// SIMATIC STEP 7 (V5.x) project jiayao
// CPU: CPU 315-2 DP
// station: P_ADR_BUS
// station: 硬件
// station: SIMATIC 300(1)(1)
// program: S7 程序(1)

SYMBOL_TABLE
"DB1"	DB 1	DB 1
"DB2"	DB 2	DB 2
"配药"	FC 1	FC 1
"计量泵程序"	FC 2	FC 2
"自动曝气"	FC 3	FC 3
"自动出药"	FC 4	FC 4
"时间转换程序"	FC 6	FC 6
"模拟液位"	FC 7	FC 7
"报警"	FC 8	FC 8
"TIM_S5TI"	FC 40	FC 40	// IEC Time to S5 Time
"SCALE"	FC 105	FC 105	// Scaling Values
"1池远程本地"	I 0.0	BOOL
"1池进药阀开到位"	I 0.1	BOOL
"1池进药阀关到位"	I 0.2	BOOL
"1池进水阀开到位"	I 0.3	BOOL
"1池进水阀关到位"	I 0.4	BOOL
"1池气阀开到位"	I 0.5	BOOL
"1池气阀关到位"	I 0.6	BOOL
"1池出药阀开到位"	I 0.7	BOOL
"1池出药阀关到位"	I 1.0	BOOL
"2池远程本地"	I 1.1	BOOL
"2池进药阀开到位"	I 1.2	BOOL
"2池进药阀关到位"	I 1.3	BOOL
"2池进水阀开到位"	I 1.4	BOOL
"2池进水阀关到位"	I 1.5	BOOL
"2池气阀开到位"	I 1.6	BOOL
"2池气阀关到位"	I 1.7	BOOL
"2池出药阀开到位"	I 2.0	BOOL
"2池出药阀关到位"	I 2.1	BOOL
"1号曝气泵远程本地"	I 2.2	BOOL
"1号曝气泵运行状态"	I 2.3	BOOL
"1号曝气泵热继故障"	I 2.4	BOOL
"2号曝气泵远程本地"	I 2.5	BOOL
"2号曝气泵运行状态"	I 2.6	BOOL
"2号曝气泵热继故障"	I 2.7	BOOL
"补水阀开到位"	I 3.0	BOOL
"新系统变频远程"	I 3.2	BOOL
"老系统变频远程"	I 3.3	BOOL
"1池自动遥控"	M 0.0	BOOL
"1池进药阀遥控开阀"	M 0.1	BOOL
"1池进药阀遥控关阀"	M 0.2	BOOL
"1池进水阀遥控开阀"	M 0.3	BOOL
"1池进水阀遥控关阀"	M 0.4	BOOL
"1池曝气阀遥控开阀"	M 0.5	BOOL
"1池曝气阀遥控关阀"	M 0.6	BOOL
"1池出药阀遥控开阀"	M 0.7	BOOL
"1池出药阀遥控关阀"	M 1.0	BOOL
"2池自动遥控"	M 1.1	BOOL
"2池进药阀遥控开阀"	M 1.2	BOOL
"2池进药阀遥控关阀"	M 1.3	BOOL
"2池进水阀遥控开阀"	M 1.4	BOOL
"2池进水阀遥控关阀"	M 1.5	BOOL
"2池进气阀遥控开阀"	M 1.6	BOOL
"2池进气阀遥控关阀"	M 1.7	BOOL
"2池出药阀遥控开阀"	M 2.0	BOOL
"2池出药阀遥控关阀"	M 2.1	BOOL
"1号曝气泵自动遥控"	M 2.2	BOOL
"1号曝气泵遥控启动"	M 2.3	BOOL
"1号曝气泵遥控停止"	M 2.4	BOOL
"2号曝气泵自动遥控"	M 2.5	BOOL
"2号曝气泵遥控启动"	M 2.6	BOOL
"2号曝气泵遥控停止"	M 2.7	BOOL
"新系统变频遥控自动"	M 3.0	BOOL
"新系统变频遥控启动"	M 3.1	BOOL
"新系统变频遥控停止"	M 3.2	BOOL
"老系统变频遥控自动"	M 3.3	BOOL
"老系统变频遥控启动"	M 3.4	BOOL
"老系统变频遥控停止"	M 3.5	BOOL
"1池空池"	M 3.6	BOOL
"2池空池"	M 3.7	BOOL
"1池确认配药"	M 4.0	BOOL
"2池确认配药"	M 4.1	BOOL
"1池取消配药"	M 4.2	BOOL
"2池取消配药"	M 4.3	BOOL
"1池开始配药"	M 4.4	BOOL
"2池开始配药"	M 4.5	BOOL
"补水阀自动遥控"	M 4.6	BOOL
"1池自动曝气系统故障"	M 4.7	BOOL
"1池气阀自动开关"	M 6.2	BOOL
"2池气阀自动开关"	M 6.3	BOOL
"配药池1号出药阀自动运行"	M 6.4	BOOL
"配药池2号出药阀自动运行"	M 6.5	BOOL
"补水阀遥控开"	M 6.6	BOOL
"补水阀遥控关"	M 6.7	BOOL
"1池气阀自动开关(延时关)"	M 7.2	BOOL
"2池气阀自动开关(延时关)"	M 7.3	BOOL
"补水阀自动开关"	M 8.6	BOOL
"1号曝气泵自动运行"	M 8.7	BOOL
"2号曝气泵自动运行"	M 9.0	BOOL
"曝气泵切换"	M 11.2	BOOL
"2.3I下降沿"	M 13.0	BOOL
"2.6I下降沿"	M 13.3	BOOL
"FC105块极性选择0为单极性"	M 15.0	BOOL
"4.4m上升沿"	M 17.1	BOOL
"1池有药"	M 17.2	BOOL
"4.5m上升沿"	M 17.3	BOOL
"2池有药"	M 17.4	BOOL
"46.6M上升沿"	M 17.5	BOOL
"47.1M上升沿"	M 17.6	BOOL
"45.0M上升沿"	M 17.7	BOOL
"1号气泵就绪"	M 18.0	BOOL
"45.1m上升沿"	M 18.1	BOOL
"2号气泵就绪"	M 18.2	BOOL
"1池计时器:运行时间上升沿"	M 18.5	BOOL
"2池计时器:运行时间上升沿"	M 18.7	BOOL
"T1计时器"	M 19.0	BOOL
"T6计时器"	M 19.1	BOOL
"1池加药阀自动运行"	M 19.2	BOOL
"1池加水阀自动运行"	M 19.3	BOOL
"2池加药阀自动运行"	M 19.4	BOOL
"2池加水阀自动运行"	M 19.5	BOOL
"1池自动曝气就绪"	M 45.0	BOOL
"2池自动曝气就绪"	M 45.1	BOOL
"2池自动曝气系统故障"	M 45.2	BOOL
"1池进药阀开故障"	M 45.3	BOOL
"1池进药阀关故障"	M 45.4	BOOL
"补水阀故障"	M 45.5	BOOL
"1池曝气请求"	M 45.6	BOOL
"2池曝气请求"	M 45.7	BOOL
"1池自动出药就绪"	M 46.0	BOOL
"1池自动出药系统故障"	M 46.1	BOOL
"1池出药阀故障"	M 46.2	BOOL
"2池自动出药系统故障"	M 46.3	BOOL
"2池自动出药就绪"	M 46.4	BOOL
"2池出药阀故障"	M 46.5	BOOL
"1池配药系统就绪"	M 46.6	BOOL
"1池配药系统故障"	M 46.7	BOOL
"2池配药系统故障"	M 47.0	BOOL
"2池配药系统就绪"	M 47.1	BOOL
"1池曝气阀故障"	M 47.2	BOOL
"2池曝气阀故障"	M 47.3	BOOL
"新系统自动运行"	M 47.4	BOOL
"1池配药"	M 47.5	BOOL
"2池配药"	M 47.6	BOOL
"老系统自动运行"	M 47.7	BOOL
"新系统变频器故障"	M 48.0	BOOL
"老系统变频器故障"	M 48.1	BOOL
"1池进药阀故障"	M 48.2	BOOL
"1池进水阀故障"	M 48.3	BOOL
"2池进药阀故障"	M 48.4	BOOL
"2池进水阀故障"	M 48.5	BOOL
"1池进水阀开故障"	M 48.6	BOOL
"1池进水阀关故障"	M 48.7	BOOL
"1池气阀开故障"	M 49.0	BOOL
"1池气阀关故障"	M 49.1	BOOL
"1池出药阀开故障"	M 49.2	BOOL
"1池出药阀关故障"	M 49.3	BOOL
"2池进药阀开故障"	M 49.4	BOOL
"2池进药阀关故障"	M 49.5	BOOL
"2池进水阀开故障"	M 49.6	BOOL
"2池进水阀关故障"	M 49.7	BOOL
"2池气阀开故障"	M 50.0	BOOL
"2池气阀关故障"	M 50.1	BOOL
"2池出药阀开故障"	M 50.2	BOOL
"2池出药阀关故障"	M 50.3	BOOL
"1号曝气泵运行故障"	M 50.4	BOOL
"2号曝气泵运行故障"	M 50.5	BOOL
"1池液位故障"	M 50.6	BOOL
"1池液位断线"	M 50.7	BOOL
"2池液位故障"	M 51.0	BOOL
"2池液位断线"	M 51.1	BOOL
"原液池液位故障"	M 51.2	BOOL
"原液池液位断线"	M 51.3	BOOL
"新系统瞬时流量下限报警"	M 51.4	BOOL	// 没用，组态已取暂留
"老系统瞬时流量下限报警"	M 51.5	BOOL	// 没用，组态已取暂留
"触摸屏消音"	M 51.6	BOOL
"COMPLETE RESTART"	OB 100	OB 100	// Complete Restart
"PROG_ERR"	OB 121	OB 121	// Programming Error
"1池进药阀开关"	Q 0.0	BOOL
"1池进水阀开关"	Q 0.1	BOOL
"1池气阀开关"	Q 0.2	BOOL
"配药池1号出药阀开关"	Q 0.3	BOOL
"2池进药阀开关"	Q 0.4	BOOL
"2池进水阀开关"	Q 0.5	BOOL
"2池气阀开关"	Q 0.6	BOOL
"配药池2号出药阀开关"	Q 0.7	BOOL
"曝气泵1号启停"	Q 1.0	BOOL
"曝气泵2号启停"	Q 1.1	BOOL
"补水阀开关"	Q 1.2	BOOL
"新系统变频启停"	Q 1.3	BOOL
"老系统变频启停"	Q 1.4	BOOL
"嗡鸣器"	Q 1.5	BOOL
"1池计时器"	T 1	TIMER
"2池计时器"	T 6	TIMER
"2池达到加药后液位"	T 7	TIMER
"2池达到加水后液位"	T 8	TIMER
"1池进药阀开故障延时"	T 9	TIMER
"1池进药阀关故障延时"	T 10	TIMER
"1池进水阀开故障延时"	T 11	TIMER
"1池进水阀关故障延时"	T 12	TIMER
"1池气阀开故障延时"	T 13	TIMER
"1池气阀关故障延时"	T 14	TIMER
"1池出药阀开故障延时"	T 15	TIMER
"1池出药阀关故障延时"	T 16	TIMER
"2池进药阀开故障延时"	T 17	TIMER
"2池进药阀关故障延时"	T 18	TIMER
"2池进水阀开故障延时"	T 19	TIMER
"2池进水阀关故障延时"	T 20	TIMER
"2池气阀开故障延时"	T 21	TIMER
"2池气阀关故障延时"	T 22	TIMER
"2池出药阀开故障延时"	T 23	TIMER
"2池出药阀关故障延时"	T 24	TIMER
"补水阀开故障延时"	T 25	TIMER
"1号曝气泵运行故障延时"	T 26	TIMER
"2号曝气泵运行故障延时"	T 27	TIMER
"1池达到加药后液位"	T 37	TIMER
"1池达到加水后液位"	T 38	TIMER
"1池曝气运行时间"	T 41	TIMER
"2池曝气运行时间"	T 42	TIMER
"新系统出药流量低延时"	T 44	TIMER
"老系统出药流量低延时"	T 45	TIMER
"1池延时断开"	T 46	TIMER
"2池延时断开"	T 47	TIMER
"1池空池延时"	T 48	TIMER
"2池空池延时"	T 49	TIMER
END_SYMBOL_TABLE

FUNCTION "配药" : VOID	// FC 1
//配药
VERSION : 0.1
BEGIN
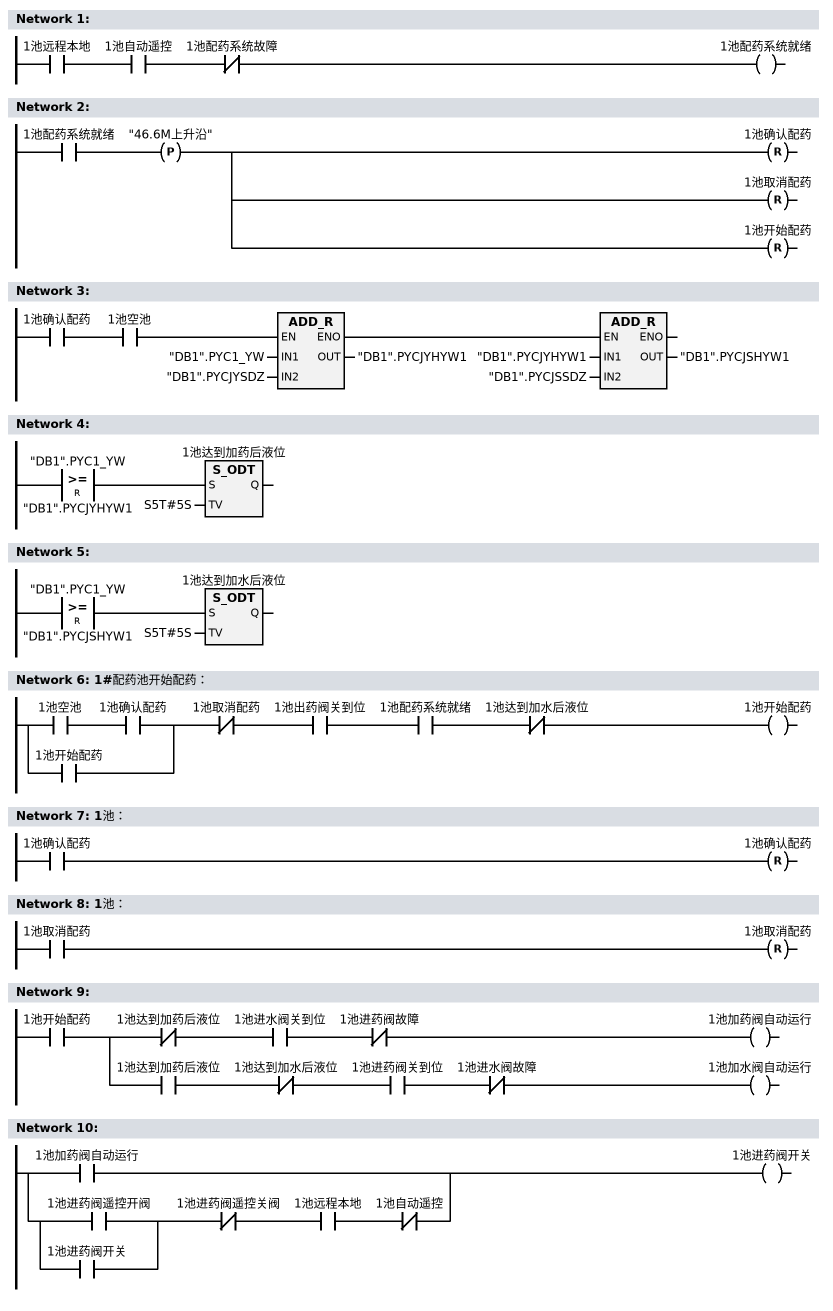
NETWORK
TITLE =
//1#配药池：配药就绪检测
      A     "1池远程本地";
      A     "1池自动遥控";
      AN    "1池配药系统故障";
      =     "1池配药系统就绪";
NETWORK
TITLE =
//1#配药池配药就绪后复位1#配药池确认、1#配药池取消配药和1#配药池开始配药
      A     "1池配药系统就绪";
      FP    "46.6M上升沿";
      R     "1池确认配药";
      R     "1池取消配药";
      R     "1池开始配药";
NETWORK
TITLE =
//1#配药池确认配药和1#配药池空池时，用1#配药池液位加上加药量设定得到1#配药池加药
//
//后的液位，用1#配药池加药后的液位加上加水量设定得到1#配药池加水后液位
      A(;
      A     "1池确认配药";
      A     "1池空池";
      JNB   _001;
      L     "DB1".PYC1_YW;
      L     "DB1".PYCJYSDZ;
      +R;
      T     "DB1".PYCJYHYW1;
      AN    OV;
      SAVE;
      CLR;
_001: A     BR;
      );
      JNB   _002;
      L     "DB1".PYCJYHYW1;
      L     "DB1".PYCJSSDZ;
      +R;
      T     "DB1".PYCJSHYW1;
_002: NOP   0;
NETWORK
TITLE =
//1#配药池液位大于等于1#加药后液位设定，延时5秒
      A(;
      L     "DB1".PYC1_YW;
      L     "DB1".PYCJYHYW1;
      >=R;
      );
      L     S5T#5S;
      SD    "1池达到加药后液位";
      NOP   0;
      NOP   0;
      NOP   0;
      NOP   0;
NETWORK
TITLE =
//1#配药池液位大于等于1#加水后液位设定，延时5秒
      A(;
      L     "DB1".PYC1_YW;
      L     "DB1".PYCJSHYW1;
      >=R;
      );
      L     S5T#5S;
      SD    "1池达到加水后液位";
      NOP   0;
      NOP   0;
      NOP   0;
      NOP   0;
NETWORK
TITLE = 1#配药池开始配药：
//
//1#配药池空池、1#配药池确认配药、1#配药池没有取消配药、1#配药池出药阀关到位、1#配
//
//药池系统就绪、1#配药池没到加水后液位，1#配药池开始配药
      A(;
      A     "1池空池";
      A     "1池确认配药";
      O     "1池开始配药";
      );
      AN    "1池取消配药";
      A     "1池出药阀关到位";
      A     "1池配药系统就绪";
      AN    "1池达到加水后液位";
      =     "1池开始配药";
NETWORK
TITLE = 1池：
//1#配药池确认配药复位
      A     "1池确认配药";
      R     "1池确认配药";
NETWORK
TITLE = 1池：
//1#配药池取消配药复位
      A     "1池取消配药";
      R     "1池取消配药";
NETWORK
TITLE =
//1#配药池开始配药，1#配药池没有达到加药后液位、1#配药池进水阀门关到位和1#配药池进
//
//药阀门无故障，1#配药池加药阀门自动运行。
//
//1#配药池开始配药，1#配药池达到加药后液位、1#配药池没有达到加水后液位、1#配药池进
//
//药阀门关到位和1#配药池进水阀门无故障，1#配药池加水阀门自动运行。
      A     "1池开始配药";
      =     L 0.0;
      A     L 0.0;
      AN    "1池达到加药后液位";
      A     "1池进水阀关到位";
      AN    "1池进药阀故障";
      =     "1池加药阀自动运行";
      A     L 0.0;
      A     "1池达到加药后液位";
      AN    "1池达到加水后液位";
      A     "1池进药阀关到位";
      AN    "1池进水阀故障";
      =     "1池加水阀自动运行";
NETWORK
TITLE =
//1#配药池进药阀自动控制和遥控控制
      O     "1池加药阀自动运行";
      O;
      A(;
      O     "1池进药阀遥控开阀";
      O     "1池进药阀开关";
      );
      AN    "1池进药阀遥控关阀";
      A     "1池远程本地";
      AN    "1池自动遥控";
      =     "1池进药阀开关";
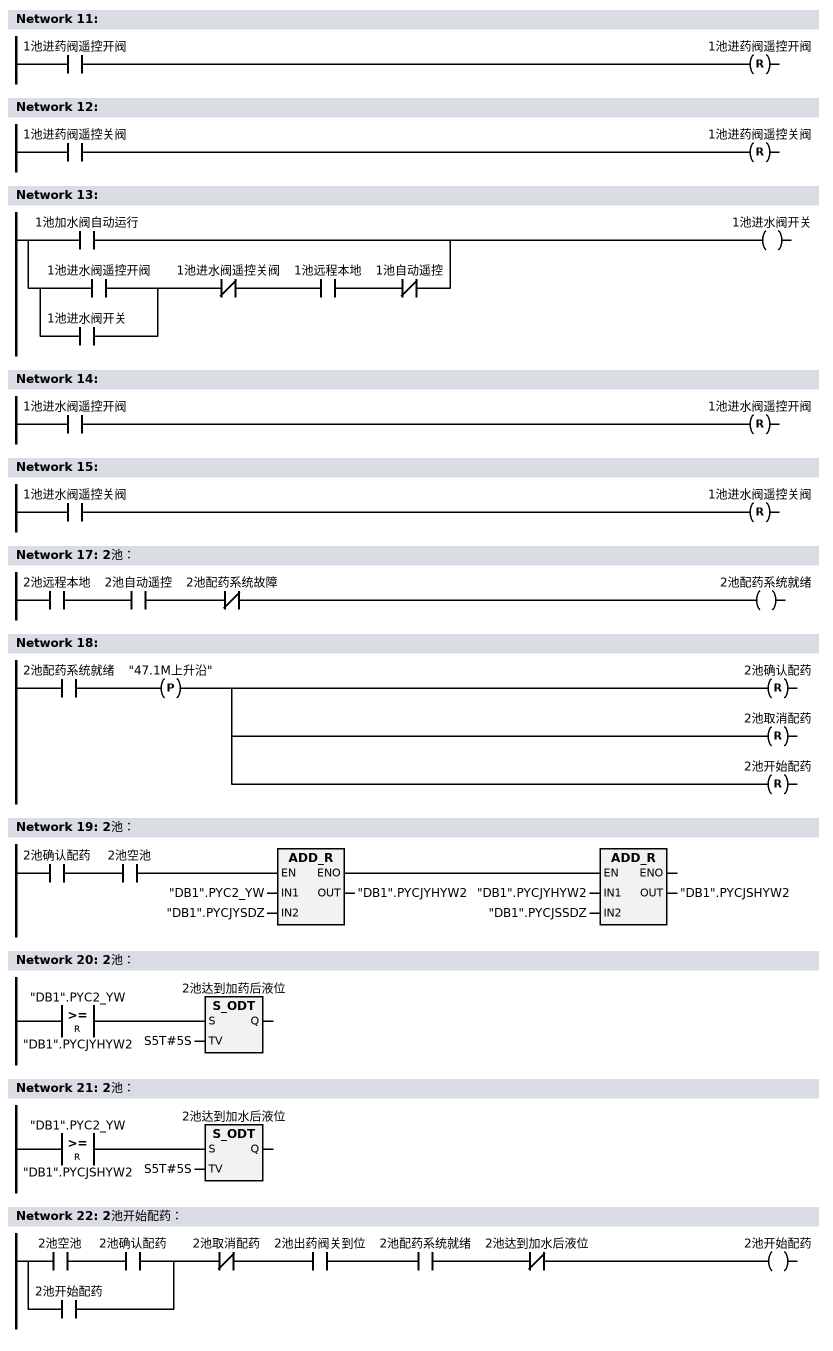
NETWORK
TITLE =
//1#配药池进药阀遥控开复位
      A     "1池进药阀遥控开阀";
      R     "1池进药阀遥控开阀";
NETWORK
TITLE =
//1#配药池进药阀遥控关复位
      A     "1池进药阀遥控关阀";
      R     "1池进药阀遥控关阀";
NETWORK
TITLE =
//1#配药池进水阀自动控制和遥控控制
      O     "1池加水阀自动运行";
      O;
      A(;
      O     "1池进水阀遥控开阀";
      O     "1池进水阀开关";
      );
      AN    "1池进水阀遥控关阀";
      A     "1池远程本地";
      AN    "1池自动遥控";
      =     "1池进水阀开关";
NETWORK
TITLE =
//1#配药池进水阀遥控开复位
      A     "1池进水阀遥控开阀";
      R     "1池进水阀遥控开阀";
NETWORK
TITLE =
//1#配药池进水阀遥控关复位
      A     "1池进水阀遥控关阀";
      R     "1池进水阀遥控关阀";
NETWORK
TITLE =
NETWORK
TITLE = 2池：
//2#配药池：配药就绪检测
      A     "2池远程本地";
      A     "2池自动遥控";
      AN    "2池配药系统故障";
      =     "2池配药系统就绪";
NETWORK
TITLE =
//2#配药池配药就绪后复位2#配药池确认、2#配药池取消配药和2#配药池开始配药
      A     "2池配药系统就绪";
      FP    "47.1M上升沿";
      R     "2池确认配药";
      R     "2池取消配药";
      R     "2池开始配药";
NETWORK
TITLE = 2池：
//2#配药池确认配药和2#配药池空池时，用2#配药池液位加上加药量设定得到2#配药池加药
//
//后的液位，用2#配药池加药后的液位加上加水量设定得到2#配药池加水后液位
      A(;
      A     "2池确认配药";
      A     "2池空池";
      JNB   _003;
      L     "DB1".PYC2_YW;
      L     "DB1".PYCJYSDZ;
      +R;
      T     "DB1".PYCJYHYW2;
      AN    OV;
      SAVE;
      CLR;
_003: A     BR;
      );
      JNB   _004;
      L     "DB1".PYCJYHYW2;
      L     "DB1".PYCJSSDZ;
      +R;
      T     "DB1".PYCJSHYW2;
_004: NOP   0;
NETWORK
TITLE = 2池：
//2#配药池液位大于等于2#加药后液位设定，延时5秒
      A(;
      L     "DB1".PYC2_YW;
      L     "DB1".PYCJYHYW2;
      >=R;
      );
      L     S5T#5S;
      SD    "2池达到加药后液位";
      NOP   0;
      NOP   0;
      NOP   0;
      NOP   0;
NETWORK
TITLE = 2池：
//2#配药池液位大于等于2#加水后液位设定，延时5秒
      A(;
      L     "DB1".PYC2_YW;
      L     "DB1".PYCJSHYW2;
      >=R;
      );
      L     S5T#5S;
      SD    "2池达到加水后液位";
      NOP   0;
      NOP   0;
      NOP   0;
      NOP   0;
NETWORK
TITLE = 2池开始配药：
//2#配药池空池、2#配药池确认配药、2#配药池没有取消配药、2#配药池出药阀关到位、2#配
//
//药池系统就绪、2#配药池没到加水后液位，2#配药池开始配药
      A(;
      A     "2池空池";
      A     "2池确认配药";
      O     "2池开始配药";
      );
      AN    "2池取消配药";
      A     "2池出药阀关到位";
      A     "2池配药系统就绪";
      AN    "2池达到加水后液位";
      =     "2池开始配药";
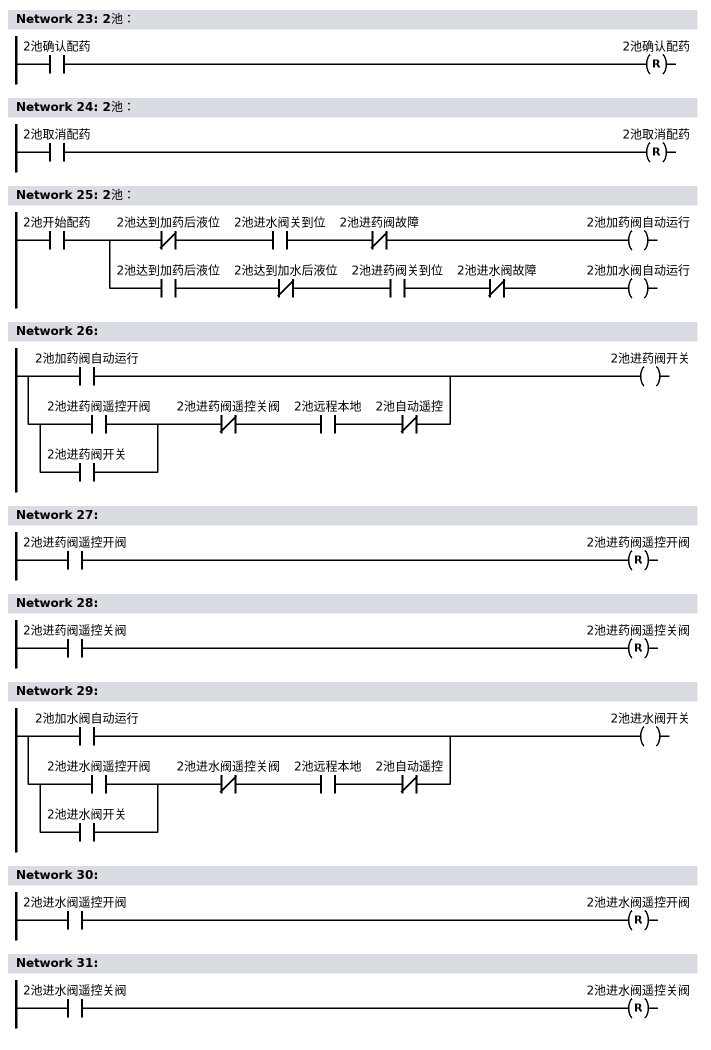
NETWORK
TITLE = 2池：
//2#配药池确认配药复位
      A     "2池确认配药";
      R     "2池确认配药";
NETWORK
TITLE = 2池：
//2#配药池取消配药复位
      A     "2池取消配药";
      R     "2池取消配药";
NETWORK
TITLE = 2池：
//2#配药池开始配药，2#配药池没有达到加药后液位、2#配药池进水阀门关到位和2#配药池进
//
//药阀门无故障，2#配药池加药阀门自动运行。
//
//2#配药池开始配药，2#配药池达到加药后液位、2#配药池没有达到加水后液位、2#配药池进
//
//药阀门关到位和2#配药池进水阀门无故障，2#配药池加水阀门自动运行
      A     "2池开始配药";
      =     L 0.0;
      A     L 0.0;
      AN    "2池达到加药后液位";
      A     "2池进水阀关到位";
      AN    "2池进药阀故障";
      =     "2池加药阀自动运行";
      A     L 0.0;
      A     "2池达到加药后液位";
      AN    "2池达到加水后液位";
      A     "2池进药阀关到位";
      AN    "2池进水阀故障";
      =     "2池加水阀自动运行";
NETWORK
TITLE =
//2#配药池进药阀自动控制和遥控控制
      O     "2池加药阀自动运行";
      O;
      A(;
      O     "2池进药阀遥控开阀";
      O     "2池进药阀开关";
      );
      AN    "2池进药阀遥控关阀";
      A     "2池远程本地";
      AN    "2池自动遥控";
      =     "2池进药阀开关";
NETWORK
TITLE =
//2#配药池进药阀遥控开复位
      A     "2池进药阀遥控开阀";
      R     "2池进药阀遥控开阀";
NETWORK
TITLE =
//2#配药池进药阀遥控关复位
      A     "2池进药阀遥控关阀";
      R     "2池进药阀遥控关阀";
NETWORK
TITLE =
//2#配药池进水阀自动控制和遥控控制
      O     "2池加水阀自动运行";
      O;
      A(;
      O     "2池进水阀遥控开阀";
      O     "2池进水阀开关";
      );
      AN    "2池进水阀遥控关阀";
      A     "2池远程本地";
      AN    "2池自动遥控";
      =     "2池进水阀开关";
NETWORK
TITLE =
//2#配药池进水阀遥控开复位
      A     "2池进水阀遥控开阀";
      R     "2池进水阀遥控开阀";
NETWORK
TITLE =
//2#配药池进水阀遥控关复位
      A     "2池进水阀遥控关阀";
      R     "2池进水阀遥控关阀";
END_FUNCTION

FUNCTION "计量泵程序" : VOID	// FC 2
//计量泵程序
VERSION : 0.1
BEGIN
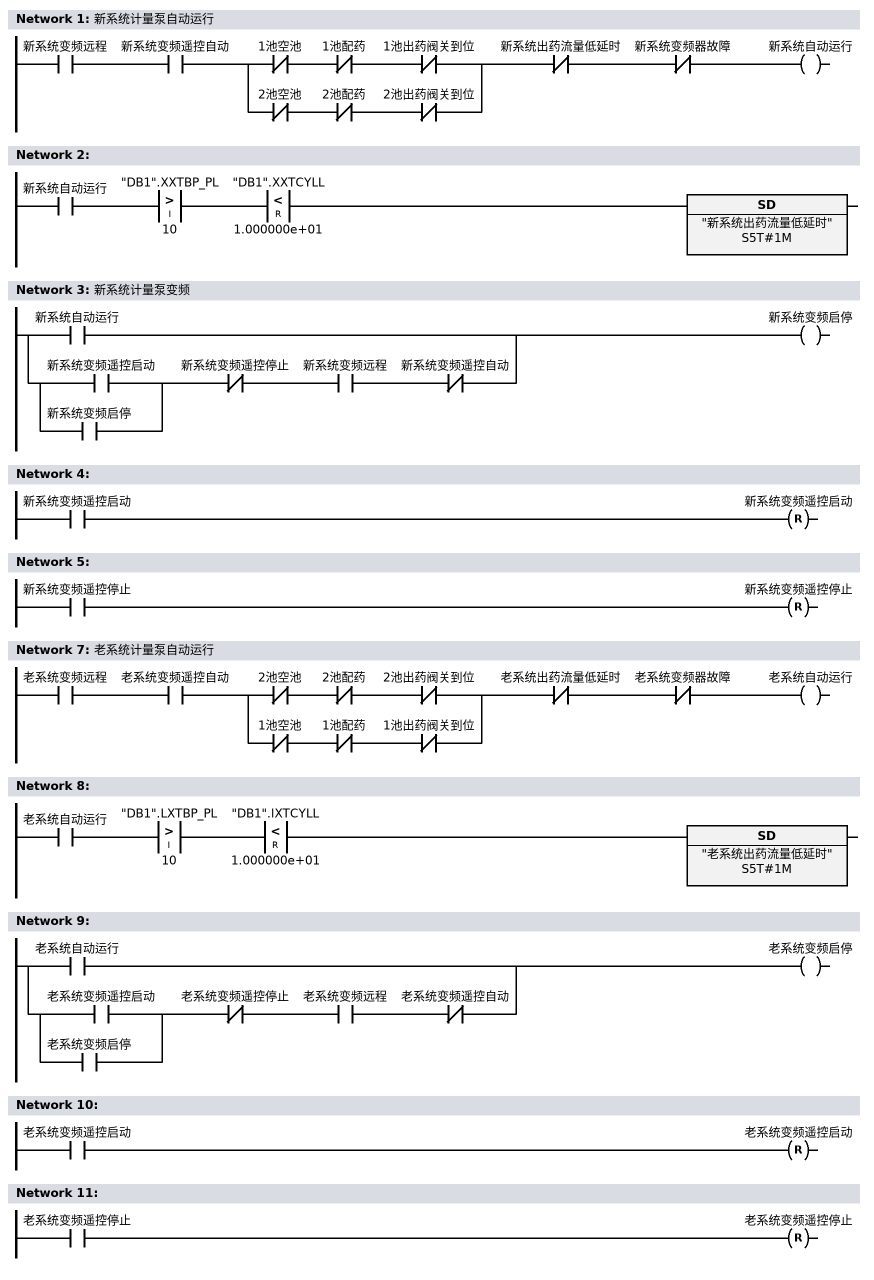
NETWORK
TITLE = 新系统计量泵自动运行
//新系统变频远程、新系统变频自动、（1#配药池不空池、1#配药池不配药、1#配药池出药阀
//
//关 或 2#配药池不空池、2#配药池不配药、2#配药池出药阀关）新系统变频出药流量不低、
//
//新系统变频无故障，新系统变频自动运行。
//
//
      A     "新系统变频远程";
      A     "新系统变频遥控自动";
      A(;
      AN    "1池空池";
      AN    "1池配药";
      AN    "1池出药阀关到位";
      O;
      AN    "2池空池";
      AN    "2池配药";
      AN    "2池出药阀关到位";
      );
      AN    "新系统出药流量低延时";
      AN    "新系统变频器故障";
      =     "新系统自动运行";
NETWORK
TITLE =
//新系统自动运行、新系统变频频率打于10和新系统瞬时流量小于10时，延时1分钟，新系统
//出药流量低
      A     "新系统自动运行";
      A(;
      L     "DB1".XXTBP_PL;
      L     10;
      >I;
      );
      A(;
      L     "DB1".XXTCYLL;
      L     1.000000e+01;
      <R;
      );
      L     S5T#1M;
      SD    "新系统出药流量低延时";
NETWORK
TITLE = 新系统计量泵变频
//新系统计量泵变频自动控制和遥控控制
      O     "新系统自动运行";
      O;
      A(;
      O     "新系统变频遥控启动";
      O     "新系统变频启停";
      );
      AN    "新系统变频遥控停止";
      A     "新系统变频远程";
      AN    "新系统变频遥控自动";
      =     "新系统变频启停";
NETWORK
TITLE =
//新系统计量泵变频遥控开复位
      A     "新系统变频遥控启动";
      R     "新系统变频遥控启动";
NETWORK
TITLE =
//新系统计量泵变频遥控关复位
      A     "新系统变频遥控停止";
      R     "新系统变频遥控停止";
NETWORK
TITLE =
NETWORK
TITLE = 老系统计量泵自动运行
//老系统变频远程、老系统变频自动、（1#配药池不空池、1#配药池不配药、1#配药池出药阀
//
//关 或 2#配药池不空池、2#配药池不配药、2#配药池出药阀关）老系统变频出药流量不低、
//
//老系统变频无故障，老系统变频自动运行。
//
      A     "老系统变频远程";
      A     "老系统变频遥控自动";
      A(;
      AN    "2池空池";
      AN    "2池配药";
      AN    "2池出药阀关到位";
      O;
      AN    "1池空池";
      AN    "1池配药";
      AN    "1池出药阀关到位";
      );
      AN    "老系统出药流量低延时";
      AN    "老系统变频器故障";
      =     "老系统自动运行";
NETWORK
TITLE =
//老系统自动运行、老系统变频频率打于10和老系统瞬时流量小于10时，延时1分钟，老系统
//出药流量低
      A     "老系统自动运行";
      A(;
      L     "DB1".LXTBP_PL;
      L     10;
      >I;
      );
      A(;
      L     "DB1".lXTCYLL;
      L     1.000000e+01;
      <R;
      );
      L     S5T#1M;
      SD    "老系统出药流量低延时";
NETWORK
TITLE =
//老系统计量泵变频自动控制和遥控控制
      O     "老系统自动运行";
      O;
      A(;
      O     "老系统变频遥控启动";
      O     "老系统变频启停";
      );
      AN    "老系统变频遥控停止";
      A     "老系统变频远程";
      AN    "老系统变频遥控自动";
      =     "老系统变频启停";
NETWORK
TITLE =
//老系统计量泵变频变频遥控开复位
      A     "老系统变频遥控启动";
      R     "老系统变频遥控启动";
NETWORK
TITLE =
//老系统计量泵变频变频遥控关复位
      A     "老系统变频遥控停止";
      R     "老系统变频遥控停止";
END_FUNCTION

FUNCTION "自动曝气" : VOID	// FC 3
//自动曝气
VERSION : 0.1
BEGIN
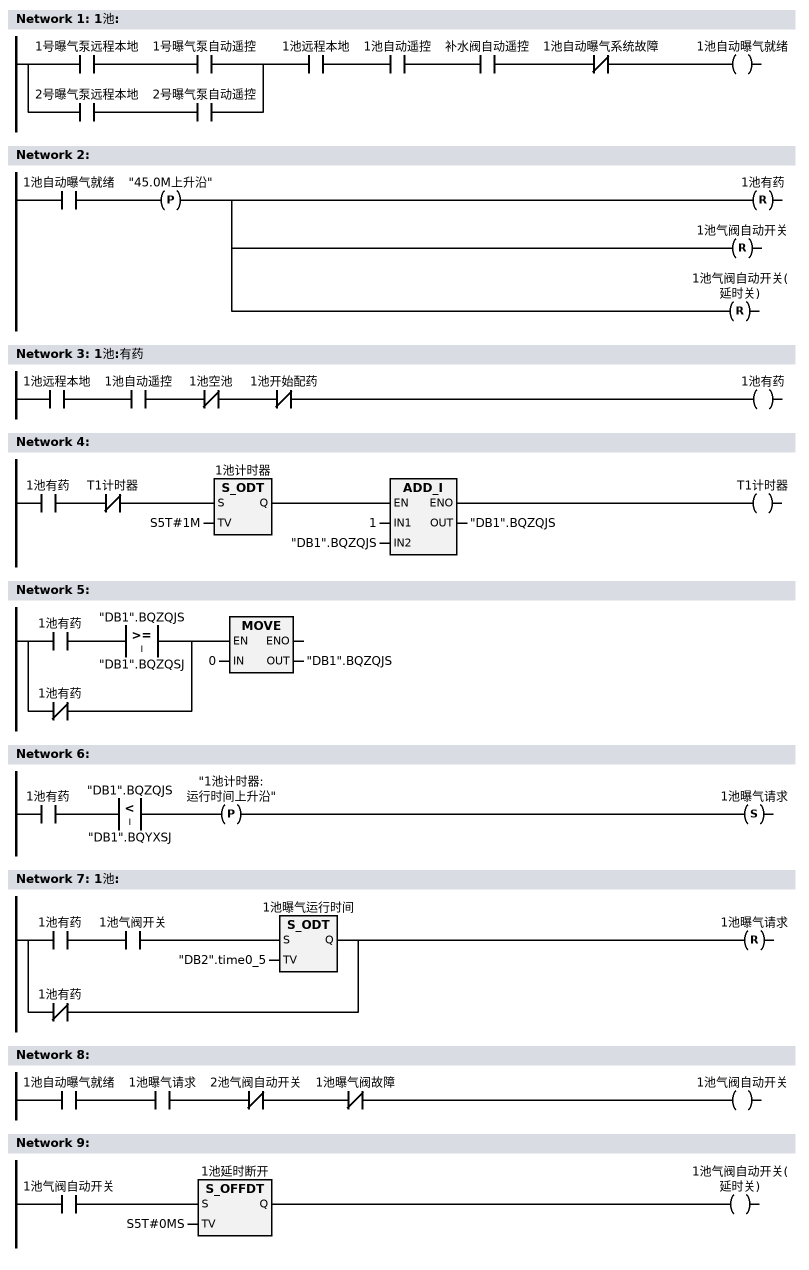
NETWORK
TITLE = 1池:
//1#配药池自动曝气就绪检测
      A(;
      A     "1号曝气泵远程本地";
      A     "1号曝气泵自动遥控";
      O;
      A     "2号曝气泵远程本地";
      A     "2号曝气泵自动遥控";
      );
      A     "1池远程本地";
      A     "1池自动遥控";
      A     "补水阀自动遥控";
      AN    "1池自动曝气系统故障";
      =     "1池自动曝气就绪";
NETWORK
TITLE =
//1#配药池自动曝气就绪后，复位1#配药池有药、1#配药池自动开关和1#配药池自动开关延时
//关
      A     "1池自动曝气就绪";
      FP    "45.0M上升沿";
      R     "1池有药";
      R     "1池气阀自动开关";
      R     "1池气阀自动开关(延时关)";
NETWORK
TITLE = 1池:有药
//1#配药池有药检测
      A     "1池远程本地";
      A     "1池自动遥控";
      AN    "1池空池";
      AN    "1池开始配药";
      =     "1池有药";
NETWORK
TITLE =
//1#配药池:曝气曝气计时器(1分钟加1)
      A(;
      A     "1池有药";
      AN    "T1计时器";
      L     S5T#1M;
      SD    "1池计时器";
      NOP   0;
      NOP   0;
      NOP   0;
      A     "1池计时器";
      );
      JNB   _001;
      L     1;
      L     "DB1".BQZQJS;
      +I;
      T     "DB1".BQZQJS;
      AN    OV;
      SAVE;
      CLR;
_001: A     BR;
      =     "T1计时器";
NETWORK
TITLE =
//1#配药池:计时器时间=周期时间或没药时计时器清零
      A(;
      A     "1池有药";
      A(;
      L     "DB1".BQZQJS;
      L     "DB1".BQZQSJ;
      >=I;
      );
      ON    "1池有药";
      );
      JNB   _002;
      L     0;
      T     "DB1".BQZQJS;
_002: NOP   0;
NETWORK
TITLE =
//1#配药池有药时、1#配药池曝气计时小于曝气运行时间设定值时上升沿，1#配药池曝气请求
//置位
      A     "1池有药";
      A(;
      L     "DB1".BQZQJS;
      L     "DB1".BQYXSJ;
      <I;
      );
      FP    "1池计时器:运行时间上升沿";
      S     "1池曝气请求";
NETWORK
TITLE = 1池:
//1#配药池有药、1#配药池气阀开和达到1#配药池曝气运行时间（运行时间上位机设定），复
//
//位1#配药池曝气请求。
//
//1#配药池没有药，复位1#配药池曝气请求。
      O(;
      A     "1池有药";
      A     "1池气阀开关";
      L     "DB2".time0_5;
      SD    "1池曝气运行时间";
      NOP   0;
      NOP   0;
      NOP   0;
      A     "1池曝气运行时间";
      );
      ON    "1池有药";
      R     "1池曝气请求";
NETWORK
TITLE =
//1配药池:曝气阀自动控制
      A     "1池自动曝气就绪";
      A     "1池曝气请求";
      AN    "2池气阀自动开关";
      AN    "1池曝气阀故障";
      =     "1池气阀自动开关";
NETWORK
TITLE =
//1#配药池:曝气阀控制M6.2断开后，延时断开M7.2
      A     "1池气阀自动开关";
      L     S5T#0MS;
      SF    "1池延时断开";
      NOP   0;
      NOP   0;
      NOP   0;
      A     "1池延时断开";
      =     "1池气阀自动开关(延时关)";
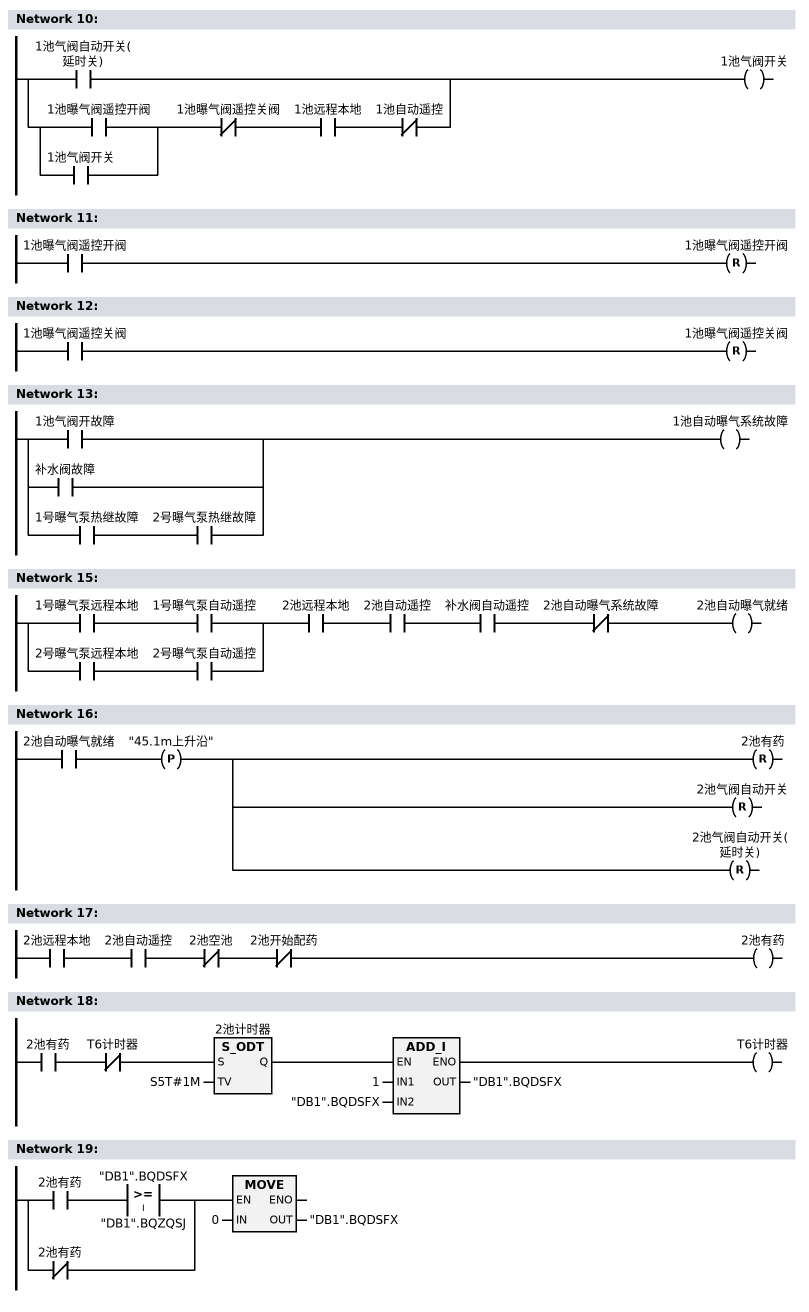
NETWORK
TITLE =
//1#配药池曝气阀自动控制和遥控控制
      O     "1池气阀自动开关(延时关)";
      O;
      A(;
      O     "1池曝气阀遥控开阀";
      O     "1池气阀开关";
      );
      AN    "1池曝气阀遥控关阀";
      A     "1池远程本地";
      AN    "1池自动遥控";
      =     "1池气阀开关";
NETWORK
TITLE =
//1#配药池曝气阀遥控开复位
      A     "1池曝气阀遥控开阀";
      R     "1池曝气阀遥控开阀";
NETWORK
TITLE =
//1#配药池曝气阀遥控关复位
      A     "1池曝气阀遥控关阀";
      R     "1池曝气阀遥控关阀";
NETWORK
TITLE =
//1池:故障检测
      O     "1池气阀开故障";
      O     "补水阀故障";
      O;
      A     "1号曝气泵热继故障";
      A     "2号曝气泵热继故障";
      =     "1池自动曝气系统故障";
NETWORK
TITLE =
NETWORK
TITLE =
//2#配药池自动曝气就绪检测
      A(;
      A     "1号曝气泵远程本地";
      A     "1号曝气泵自动遥控";
      O;
      A     "2号曝气泵远程本地";
      A     "2号曝气泵自动遥控";
      );
      A     "2池远程本地";
      A     "2池自动遥控";
      A     "补水阀自动遥控";
      AN    "2池自动曝气系统故障";
      =     "2池自动曝气就绪";
NETWORK
TITLE =
//2#配药池自动曝气就绪后，复位2#配药池有药、2#配药池自动开关和2#配药池自动开关延时
//关
      A     "2池自动曝气就绪";
      FP    "45.1m上升沿";
      R     "2池有药";
      R     "2池气阀自动开关";
      R     "2池气阀自动开关(延时关)";
NETWORK
TITLE =
//2#配药池有药检测
      A     "2池远程本地";
      A     "2池自动遥控";
      AN    "2池空池";
      AN    "2池开始配药";
      =     "2池有药";
NETWORK
TITLE =
//2#配药池:曝气曝气计时器(1分钟加1)
      A(;
      A     "2池有药";
      AN    "T6计时器";
      L     S5T#1M;
      SD    "2池计时器";
      NOP   0;
      NOP   0;
      NOP   0;
      A     "2池计时器";
      );
      JNB   _003;
      L     1;
      L     "DB1".BQDSFX;
      +I;
      T     "DB1".BQDSFX;
      AN    OV;
      SAVE;
      CLR;
_003: A     BR;
      =     "T6计时器";
NETWORK
TITLE =
//2#配药池:计时器时间=周期时间或没药时计时器清零
      A(;
      A     "2池有药";
      A(;
      L     "DB1".BQDSFX;
      L     "DB1".BQZQSJ;
      >=I;
      );
      ON    "2池有药";
      );
      JNB   _004;
      L     0;
      T     "DB1".BQDSFX;
_004: NOP   0;
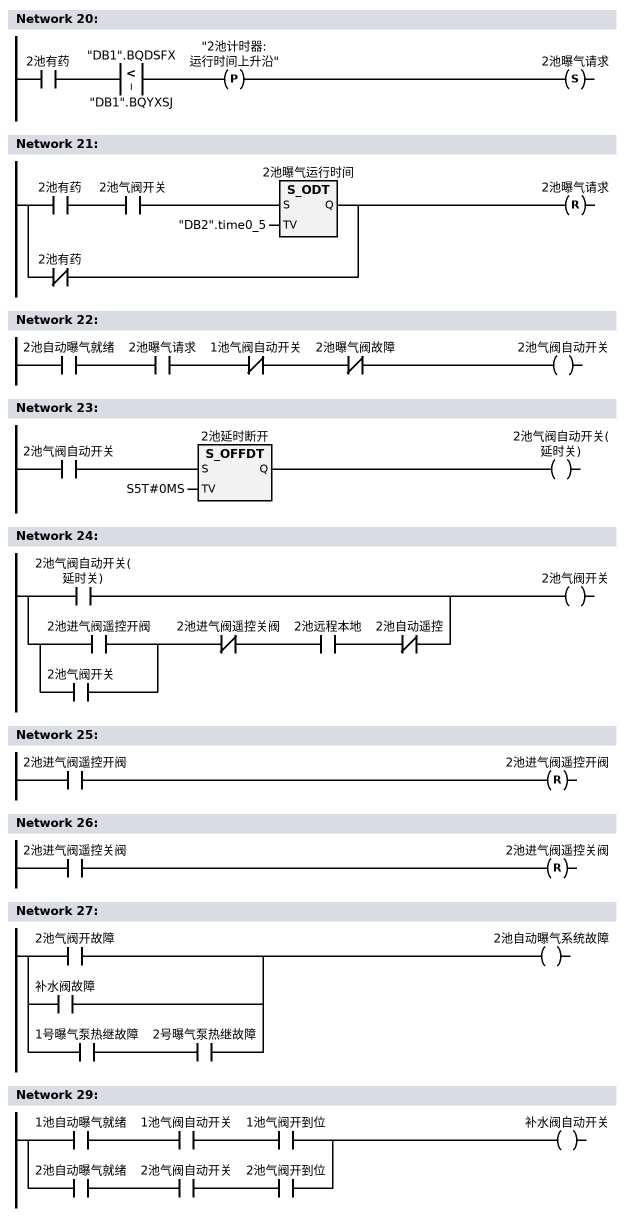
NETWORK
TITLE =
//2#配药池有药时、2#配药池曝气计时小于曝气运行时间设定值时上升沿，2#配药池曝气请求
//置位
      A     "2池有药";
      A(;
      L     "DB1".BQDSFX;
      L     "DB1".BQYXSJ;
      <I;
      );
      FP    "2池计时器:运行时间上升沿";
      S     "2池曝气请求";
NETWORK
TITLE =
//2#配药池有药、2#配药池气阀开和达到2#配药池曝气运行时间（运行时间上位机设定），复
//
//位2#配药池曝气请求。
//
//2#配药池没有药，复位1#配药池曝气请求。
      O(;
      A     "2池有药";
      A     "2池气阀开关";
      L     "DB2".time0_5;
      SD    "2池曝气运行时间";
      NOP   0;
      NOP   0;
      NOP   0;
      A     "2池曝气运行时间";
      );
      ON    "2池有药";
      R     "2池曝气请求";
NETWORK
TITLE =
//2#配药池曝气阀自动控制
      A     "2池自动曝气就绪";
      A     "2池曝气请求";
      AN    "1池气阀自动开关";
      AN    "2池曝气阀故障";
      =     "2池气阀自动开关";
NETWORK
TITLE =
//2#配药池:曝气阀控制M6.2断开后，延时断开M7.2
      A     "2池气阀自动开关";
      L     S5T#0MS;
      SF    "2池延时断开";
      NOP   0;
      NOP   0;
      NOP   0;
      A     "2池延时断开";
      =     "2池气阀自动开关(延时关)";
NETWORK
TITLE =
//2#配药池曝气阀自动控制和遥控控制
      O     "2池气阀自动开关(延时关)";
      O;
      A(;
      O     "2池进气阀遥控开阀";
      O     "2池气阀开关";
      );
      AN    "2池进气阀遥控关阀";
      A     "2池远程本地";
      AN    "2池自动遥控";
      =     "2池气阀开关";
NETWORK
TITLE =
//2#配药池曝气阀遥控开复位
      A     "2池进气阀遥控开阀";
      R     "2池进气阀遥控开阀";
NETWORK
TITLE =
//2#配药池曝气阀遥控关复位
      A     "2池进气阀遥控关阀";
      R     "2池进气阀遥控关阀";
NETWORK
TITLE =
//2配药池:故障检测
      O     "2池气阀开故障";
      O     "补水阀故障";
      O;
      A     "1号曝气泵热继故障";
      A     "2号曝气泵热继故障";
      =     "2池自动曝气系统故障";
NETWORK
TITLE =
NETWORK
TITLE =
//补水阀自动开关
      A     "1池自动曝气就绪";
      A     "1池气阀自动开关";
      A     "1池气阀开到位";
      O;
      A     "2池自动曝气就绪";
      A     "2池气阀自动开关";
      A     "2池气阀开到位";
      =     "补水阀自动开关";
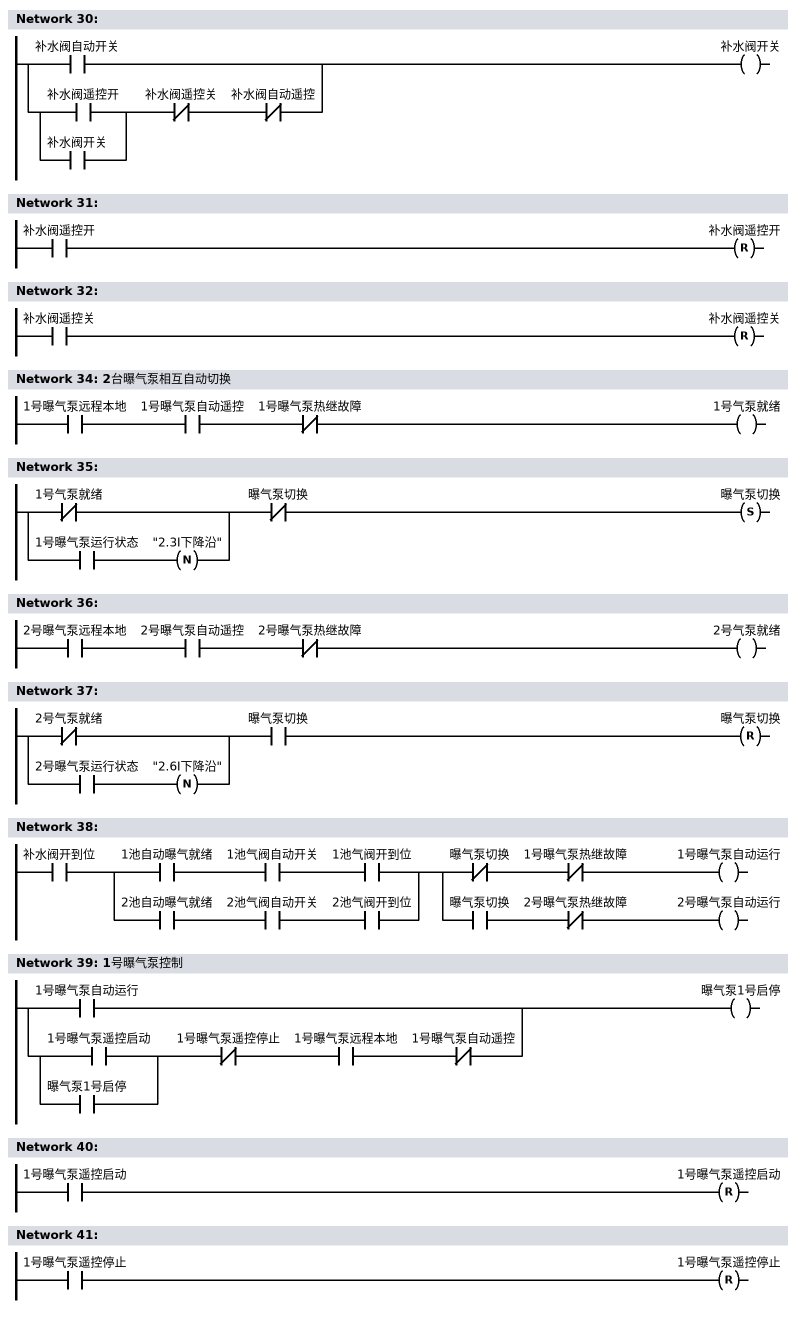
NETWORK
TITLE =
//补水阀自动开关控制和遥控开关控制
      O     "补水阀自动开关";
      O;
      A(;
      O     "补水阀遥控开";
      O     "补水阀开关";
      );
      AN    "补水阀遥控关";
      AN    "补水阀自动遥控";
      =     "补水阀开关";
NETWORK
TITLE =
//补水阀遥控开复位
      A     "补水阀遥控开";
      R     "补水阀遥控开";
NETWORK
TITLE =
//补水阀遥控关复位
      A     "补水阀遥控关";
      R     "补水阀遥控关";
NETWORK
TITLE =
NETWORK
TITLE = 2台曝气泵相互自动切换  
//1#曝气泵就绪检测
      A     "1号曝气泵远程本地";
      A     "1号曝气泵自动遥控";
      AN    "1号曝气泵热继故障";
      =     "1号气泵就绪";
NETWORK
TITLE =
//1#曝气泵没就绪或运行停止切换曝气泵
      A(;
      ON    "1号气泵就绪";
      O(;
      A     "1号曝气泵运行状态";
      FN    "2.3I下降沿";
      );
      );
      AN    "曝气泵切换";
      S     "曝气泵切换";
NETWORK
TITLE =
//2#曝气泵就绪检测
      A     "2号曝气泵远程本地";
      A     "2号曝气泵自动遥控";
      AN    "2号曝气泵热继故障";
      =     "2号气泵就绪";
NETWORK
TITLE =
//2#曝气泵没就绪或运行停止切换曝气泵
      A(;
      ON    "2号气泵就绪";
      O(;
      A     "2号曝气泵运行状态";
      FN    "2.6I下降沿";
      );
      );
      A     "曝气泵切换";
      R     "曝气泵切换";
NETWORK
TITLE =
//1#曝气泵和2#曝气泵相互自动切换运行。    m11.2是2台曝气泵相互自动切换  
      A     "补水阀开到位";
      A(;
      A     "1池自动曝气就绪";
      A     "1池气阀自动开关";
      A     "1池气阀开到位";
      O;
      A     "2池自动曝气就绪";
      A     "2池气阀自动开关";
      A     "2池气阀开到位";
      );
      =     L 0.0;
      A     L 0.0;
      AN    "曝气泵切换";
      AN    "1号曝气泵热继故障";
      =     "1号曝气泵自动运行";
      A     L 0.0;
      A     "曝气泵切换";
      AN    "2号曝气泵热继故障";
      =     "2号曝气泵自动运行";
NETWORK
TITLE = 1号曝气泵控制
//1号曝气泵自动控制和遥控控制
      O     "1号曝气泵自动运行";
      O;
      A(;
      O     "1号曝气泵遥控启动";
      O     "曝气泵1号启停";
      );
      AN    "1号曝气泵遥控停止";
      A     "1号曝气泵远程本地";
      AN    "1号曝气泵自动遥控";
      =     "曝气泵1号启停";
NETWORK
TITLE =
//1号曝气泵开复位
      A     "1号曝气泵遥控启动";
      R     "1号曝气泵遥控启动";
NETWORK
TITLE =
//1号曝气泵关复位
      A     "1号曝气泵遥控停止";
      R     "1号曝气泵遥控停止";
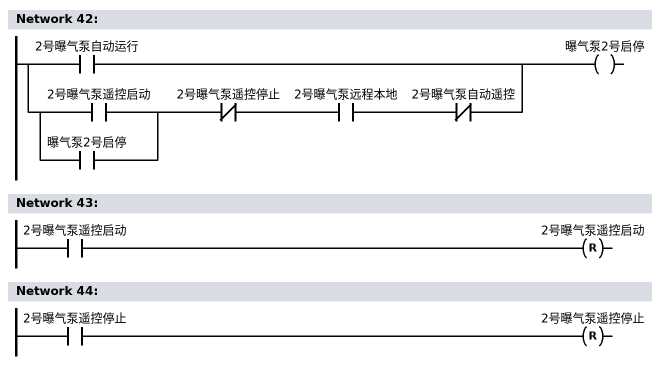
NETWORK
TITLE =
//2号曝气泵自动控制和遥控控制
      O     "2号曝气泵自动运行";
      O;
      A(;
      O     "2号曝气泵遥控启动";
      O     "曝气泵2号启停";
      );
      AN    "2号曝气泵遥控停止";
      A     "2号曝气泵远程本地";
      AN    "2号曝气泵自动遥控";
      =     "曝气泵2号启停";
NETWORK
TITLE =
//2号曝气泵开复位
      A     "2号曝气泵遥控启动";
      R     "2号曝气泵遥控启动";
NETWORK
TITLE =
//2号曝气泵关复位
      A     "2号曝气泵遥控停止";
      R     "2号曝气泵遥控停止";
END_FUNCTION

FUNCTION "自动出药" : VOID	// FC 4
//出药阀程序
VERSION : 0.1
BEGIN
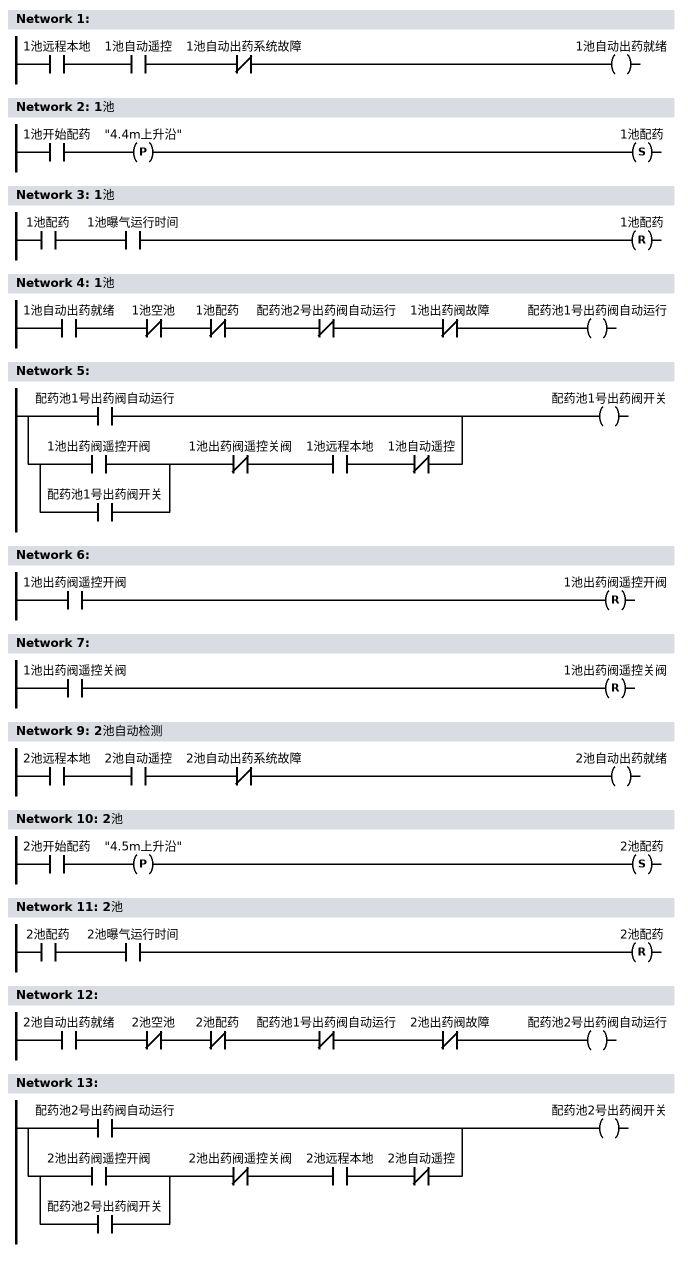
NETWORK
TITLE =
//1#配药池自动出药就绪检测
      A     "1池远程本地";
      A     "1池自动遥控";
      AN    "1池自动出药系统故障";
      =     "1池自动出药就绪";
NETWORK
TITLE = 1池
//1#配药池开始配药
      A     "1池开始配药";
      FP    "4.4m上升沿";
      S     "1池配药";
NETWORK
TITLE = 1池
//1#配药池曝气时不配药
      A     "1池配药";
      A     "1池曝气运行时间";
      R     "1池配药";
NETWORK
TITLE = 1池
//1#配药池出药阀就绪、1#配药池不空池、1#配药池没配药、2#配药池出药阀没开、1#配药池
//出药阀无故障、1#配药池出药阀自动运行。
      A     "1池自动出药就绪";
      AN    "1池空池";
      AN    "1池配药";
      AN    "配药池2号出药阀自动运行";
      AN    "1池出药阀故障";
      =     "配药池1号出药阀自动运行";
NETWORK
TITLE =
//1#配药池出药阀自动控制和遥控控制
      O     "配药池1号出药阀自动运行";
      O;
      A(;
      O     "1池出药阀遥控开阀";
      O     "配药池1号出药阀开关";
      );
      AN    "1池出药阀遥控关阀";
      A     "1池远程本地";
      AN    "1池自动遥控";
      =     "配药池1号出药阀开关";
NETWORK
TITLE =
//1#配药池池出药阀遥控开复位
      A     "1池出药阀遥控开阀";
      R     "1池出药阀遥控开阀";
NETWORK
TITLE =
//1#配药池出药阀遥控关复位
      A     "1池出药阀遥控关阀";
      R     "1池出药阀遥控关阀";
NETWORK
TITLE =
NETWORK
TITLE = 2池自动检测
//2#配药池自动出药就绪检测
      A     "2池远程本地";
      A     "2池自动遥控";
      AN    "2池自动出药系统故障";
      =     "2池自动出药就绪";
NETWORK
TITLE = 2池
//2#配药池开始配药
      A     "2池开始配药";
      FP    "4.5m上升沿";
      S     "2池配药";
NETWORK
TITLE = 2池
//2#配药池曝气时不配药
      A     "2池配药";
      A     "2池曝气运行时间";
      R     "2池配药";
NETWORK
TITLE =
//2#配药池出药阀就绪、2#配药池不空池、2#配药池没配药、1#配药池出药阀没开、2#配药池
//出药阀无故障、2#配药池出药阀自动运行。
      A     "2池自动出药就绪";
      AN    "2池空池";
      AN    "2池配药";
      AN    "配药池1号出药阀自动运行";
      AN    "2池出药阀故障";
      =     "配药池2号出药阀自动运行";
NETWORK
TITLE =
//2#配药池出药阀自动控制和遥控控制
      O     "配药池2号出药阀自动运行";
      O;
      A(;
      O     "2池出药阀遥控开阀";
      O     "配药池2号出药阀开关";
      );
      AN    "2池出药阀遥控关阀";
      A     "2池远程本地";
      AN    "2池自动遥控";
      =     "配药池2号出药阀开关";
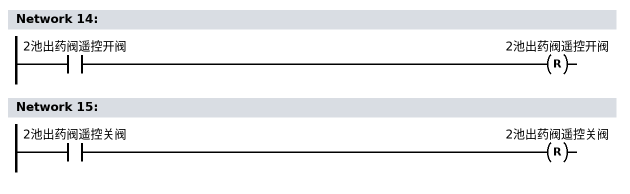
NETWORK
TITLE =
//2#配药池出药阀遥控开复位
      A     "2池出药阀遥控开阀";
      R     "2池出药阀遥控开阀";
NETWORK
TITLE =
//2#配药池出药阀遥控关复位
      A     "2池出药阀遥控关阀";
      R     "2池出药阀遥控关阀";
END_FUNCTION

FUNCTION "时间转换程序" : VOID	// FC 6
//时间转换程序
VERSION : 0.1
BEGIN
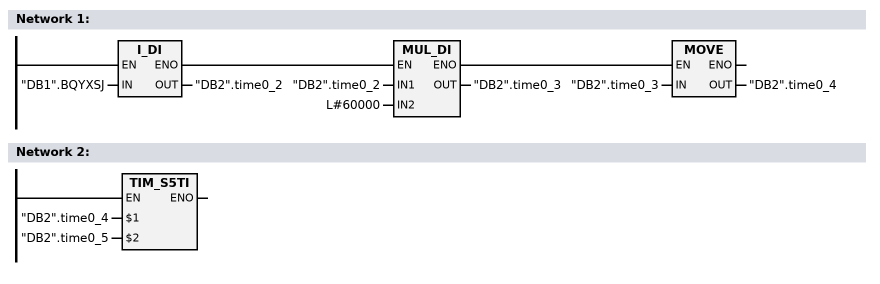
NETWORK
TITLE =
      A(;
      A(;
      L     "DB1".BQYXSJ;
      ITD;
      T     "DB2".time0_2;
      SET;
      SAVE;
      CLR;
      A     BR;
      );
      JNB   _001;
      L     "DB2".time0_2;
      L     L#60000;
      *D;
      T     "DB2".time0_3;
      AN    OV;
      SAVE;
      CLR;
_001: A     BR;
      );
      JNB   _002;
      L     "DB2".time0_3;
      T     "DB2".time0_4;
_002: NOP   0;
NETWORK
TITLE =
//把TIME格式转换成S5TIME格式
      CALL  "TIM_S5TI" (
           $1                       := "DB2".time0_4,
           $2                       := "DB2".time0_5);
      NOP   0;
NETWORK
TITLE =
NETWORK
TITLE =
NETWORK
TITLE =
END_FUNCTION

FUNCTION "报警" : VOID	// FC 8
//故障
VERSION : 0.1
BEGIN
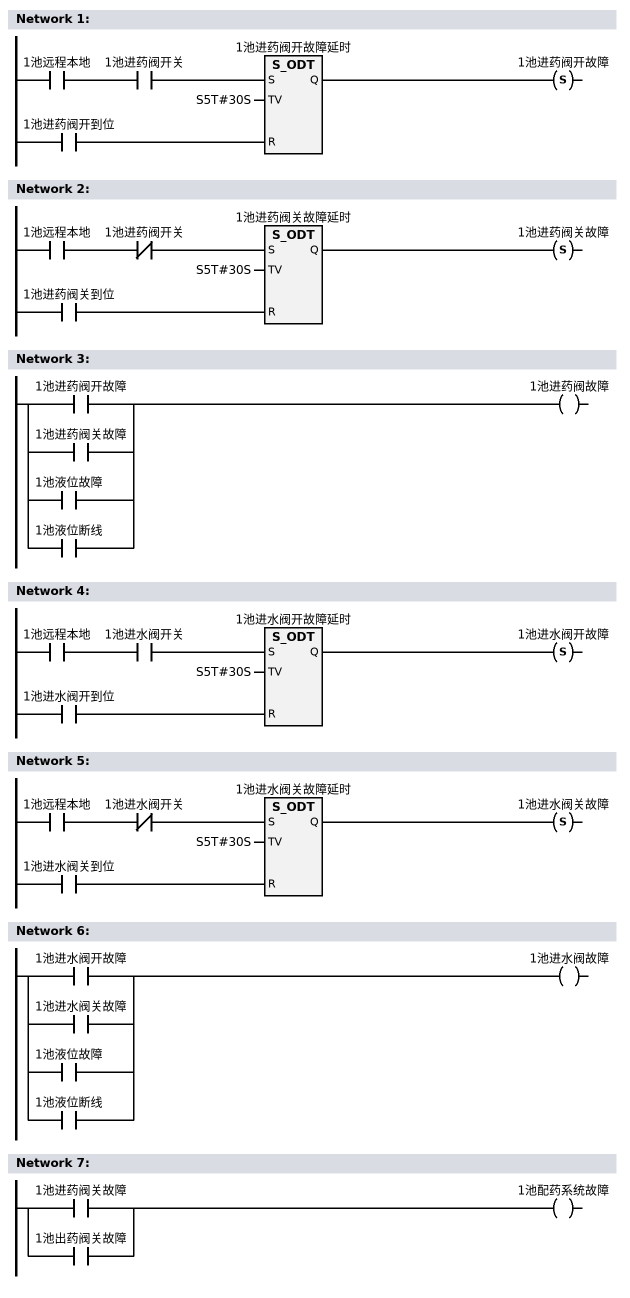
NETWORK
TITLE =
//1池进药阀开故障（30秒阀门没开到位）
      A     "1池远程本地";
      A     "1池进药阀开关";
      L     S5T#30S;
      SD    "1池进药阀开故障延时";
      A     "1池进药阀开到位";
      R     "1池进药阀开故障延时";
      NOP   0;
      NOP   0;
      A     "1池进药阀开故障延时";
      S     "1池进药阀开故障";
NETWORK
TITLE =
//1池进药阀关故障（30秒阀门没关到位）
      A     "1池远程本地";
      AN    "1池进药阀开关";
      L     S5T#30S;
      SD    "1池进药阀关故障延时";
      A     "1池进药阀关到位";
      R     "1池进药阀关故障延时";
      NOP   0;
      NOP   0;
      A     "1池进药阀关故障延时";
      S     "1池进药阀关故障";
NETWORK
TITLE =
//1池进药阀故障
      O     "1池进药阀开故障";
      O     "1池进药阀关故障";
      O     "1池液位故障";
      O     "1池液位断线";
      =     "1池进药阀故障";
NETWORK
TITLE =
//1池进水阀开故障（30秒阀门没开到位）
      A     "1池远程本地";
      A     "1池进水阀开关";
      L     S5T#30S;
      SD    "1池进水阀开故障延时";
      A     "1池进水阀开到位";
      R     "1池进水阀开故障延时";
      NOP   0;
      NOP   0;
      A     "1池进水阀开故障延时";
      S     "1池进水阀开故障";
NETWORK
TITLE =
//1池进水阀关故障（30秒阀门没关到位）
      A     "1池远程本地";
      AN    "1池进水阀开关";
      L     S5T#30S;
      SD    "1池进水阀关故障延时";
      A     "1池进水阀关到位";
      R     "1池进水阀关故障延时";
      NOP   0;
      NOP   0;
      A     "1池进水阀关故障延时";
      S     "1池进水阀关故障";
NETWORK
TITLE =
//1池进水阀故障
      O     "1池进水阀开故障";
      O     "1池进水阀关故障";
      O     "1池液位故障";
      O     "1池液位断线";
      =     "1池进水阀故障";
NETWORK
TITLE =
//1池配药系统故障
      O     "1池进药阀关故障";
      O     "1池出药阀关故障";
      =     "1池配药系统故障";
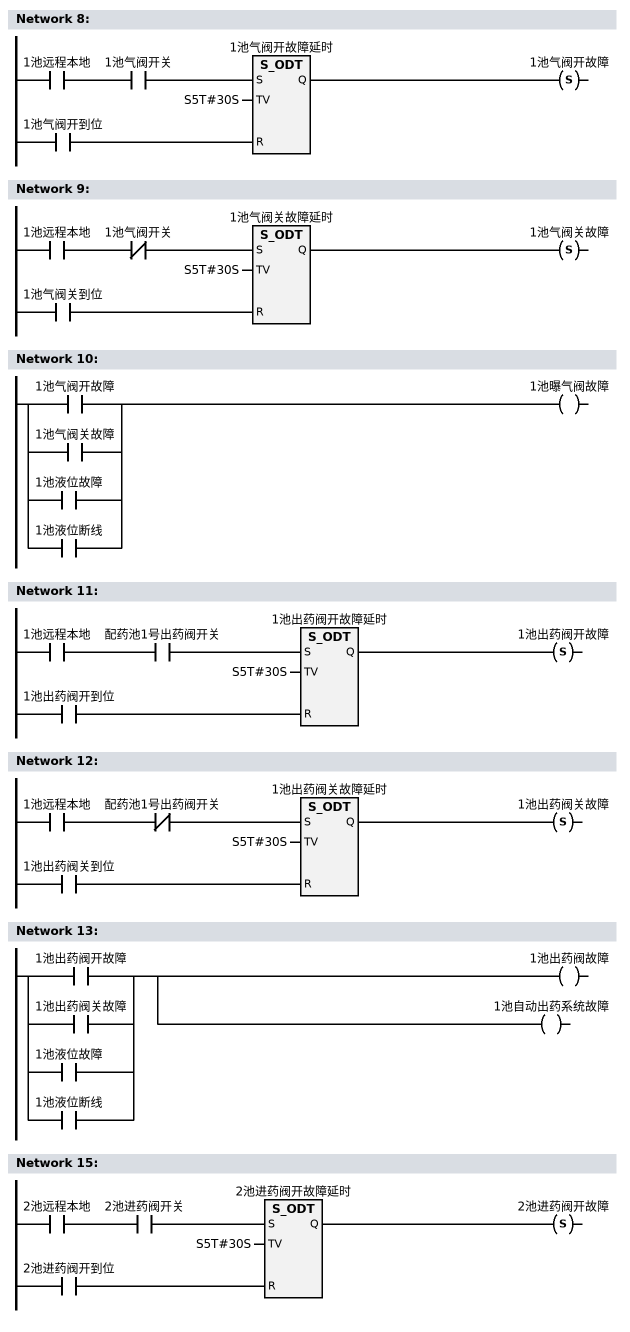
NETWORK
TITLE =
//1池气阀开故障（30秒阀门没开到位）
      A     "1池远程本地";
      A     "1池气阀开关";
      L     S5T#30S;
      SD    "1池气阀开故障延时";
      A     "1池气阀开到位";
      R     "1池气阀开故障延时";
      NOP   0;
      NOP   0;
      A     "1池气阀开故障延时";
      S     "1池气阀开故障";
NETWORK
TITLE =
//1池气阀关故障（30秒阀门没关到位）
      A     "1池远程本地";
      AN    "1池气阀开关";
      L     S5T#30S;
      SD    "1池气阀关故障延时";
      A     "1池气阀关到位";
      R     "1池气阀关故障延时";
      NOP   0;
      NOP   0;
      A     "1池气阀关故障延时";
      S     "1池气阀关故障";
NETWORK
TITLE =
//1池气阀故障
      O     "1池气阀开故障";
      O     "1池气阀关故障";
      O     "1池液位故障";
      O     "1池液位断线";
      =     "1池曝气阀故障";
NETWORK
TITLE =
//1池出药阀开故障（30秒阀门没开到位）
      A     "1池远程本地";
      A     "配药池1号出药阀开关";
      L     S5T#30S;
      SD    "1池出药阀开故障延时";
      A     "1池出药阀开到位";
      R     "1池出药阀开故障延时";
      NOP   0;
      NOP   0;
      A     "1池出药阀开故障延时";
      S     "1池出药阀开故障";
NETWORK
TITLE =
//1池出药阀关故障（30秒阀门没关到位）
      A     "1池远程本地";
      AN    "配药池1号出药阀开关";
      L     S5T#30S;
      SD    "1池出药阀关故障延时";
      A     "1池出药阀关到位";
      R     "1池出药阀关故障延时";
      NOP   0;
      NOP   0;
      A     "1池出药阀关故障延时";
      S     "1池出药阀关故障";
NETWORK
TITLE =
//1池出药阀故障
      O     "1池出药阀开故障";
      O     "1池出药阀关故障";
      O     "1池液位故障";
      O     "1池液位断线";
      =     "1池出药阀故障";
      =     "1池自动出药系统故障";
NETWORK
TITLE =
NETWORK
TITLE =
//2池进药阀开故障（30秒阀门没开到位）
      A     "2池远程本地";
      A     "2池进药阀开关";
      L     S5T#30S;
      SD    "2池进药阀开故障延时";
      A     "2池进药阀开到位";
      R     "2池进药阀开故障延时";
      NOP   0;
      NOP   0;
      A     "2池进药阀开故障延时";
      S     "2池进药阀开故障";
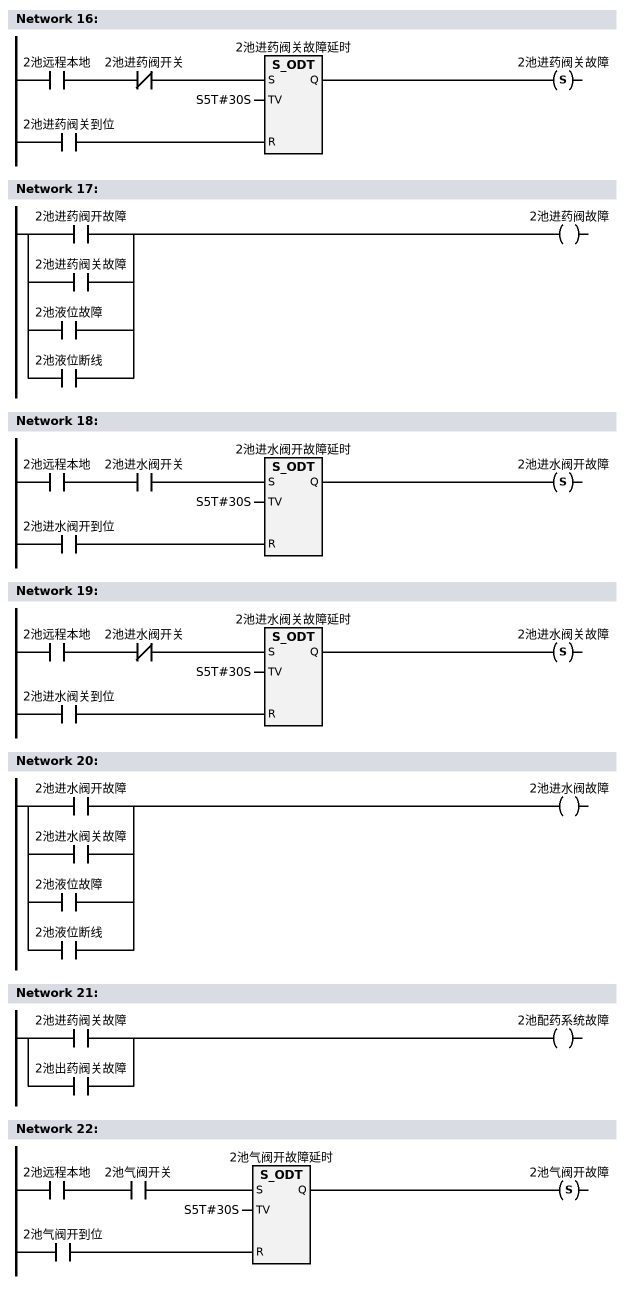
NETWORK
TITLE =
//2池进药阀关故障（30秒阀门没关到位）
      A     "2池远程本地";
      AN    "2池进药阀开关";
      L     S5T#30S;
      SD    "2池进药阀关故障延时";
      A     "2池进药阀关到位";
      R     "2池进药阀关故障延时";
      NOP   0;
      NOP   0;
      A     "2池进药阀关故障延时";
      S     "2池进药阀关故障";
NETWORK
TITLE =
//2池进药阀故障
      O     "2池进药阀开故障";
      O     "2池进药阀关故障";
      O     "2池液位故障";
      O     "2池液位断线";
      =     "2池进药阀故障";
NETWORK
TITLE =
//2池进水阀开故障（30秒阀门没开到位）
      A     "2池远程本地";
      A     "2池进水阀开关";
      L     S5T#30S;
      SD    "2池进水阀开故障延时";
      A     "2池进水阀开到位";
      R     "2池进水阀开故障延时";
      NOP   0;
      NOP   0;
      A     "2池进水阀开故障延时";
      S     "2池进水阀开故障";
NETWORK
TITLE =
//2池进水阀关故障（30秒阀门没关到位）
      A     "2池远程本地";
      AN    "2池进水阀开关";
      L     S5T#30S;
      SD    "2池进水阀关故障延时";
      A     "2池进水阀关到位";
      R     "2池进水阀关故障延时";
      NOP   0;
      NOP   0;
      A     "2池进水阀关故障延时";
      S     "2池进水阀关故障";
NETWORK
TITLE =
//2池进水阀故障
      O     "2池进水阀开故障";
      O     "2池进水阀关故障";
      O     "2池液位故障";
      O     "2池液位断线";
      =     "2池进水阀故障";
NETWORK
TITLE =
//2池配药系统故障
      O     "2池进药阀关故障";
      O     "2池出药阀关故障";
      =     "2池配药系统故障";
NETWORK
TITLE =
//2池气阀开故障（30秒阀门没开到位）
      A     "2池远程本地";
      A     "2池气阀开关";
      L     S5T#30S;
      SD    "2池气阀开故障延时";
      A     "2池气阀开到位";
      R     "2池气阀开故障延时";
      NOP   0;
      NOP   0;
      A     "2池气阀开故障延时";
      S     "2池气阀开故障";
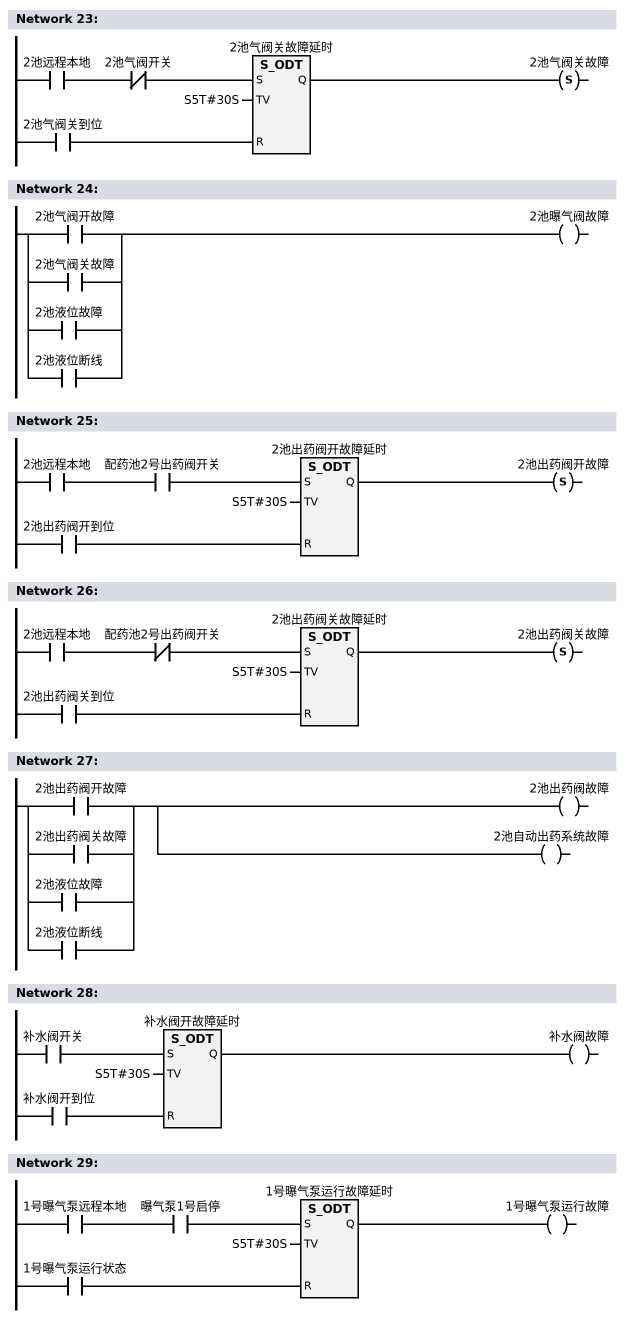
NETWORK
TITLE =
//2池气阀关故障（30秒阀门没关到位）
      A     "2池远程本地";
      AN    "2池气阀开关";
      L     S5T#30S;
      SD    "2池气阀关故障延时";
      A     "2池气阀关到位";
      R     "2池气阀关故障延时";
      NOP   0;
      NOP   0;
      A     "2池气阀关故障延时";
      S     "2池气阀关故障";
NETWORK
TITLE =
//2池气阀故障
      O     "2池气阀开故障";
      O     "2池气阀关故障";
      O     "2池液位故障";
      O     "2池液位断线";
      =     "2池曝气阀故障";
NETWORK
TITLE =
//2池出药阀开故障（30秒阀门没开到位）
      A     "2池远程本地";
      A     "配药池2号出药阀开关";
      L     S5T#30S;
      SD    "2池出药阀开故障延时";
      A     "2池出药阀开到位";
      R     "2池出药阀开故障延时";
      NOP   0;
      NOP   0;
      A     "2池出药阀开故障延时";
      S     "2池出药阀开故障";
NETWORK
TITLE =
//2池出药阀关故障（30秒阀门没关到位）
      A     "2池远程本地";
      AN    "配药池2号出药阀开关";
      L     S5T#30S;
      SD    "2池出药阀关故障延时";
      A     "2池出药阀关到位";
      R     "2池出药阀关故障延时";
      NOP   0;
      NOP   0;
      A     "2池出药阀关故障延时";
      S     "2池出药阀关故障";
NETWORK
TITLE =
//2池出药阀故障
      O     "2池出药阀开故障";
      O     "2池出药阀关故障";
      O     "2池液位故障";
      O     "2池液位断线";
      =     "2池出药阀故障";
      =     "2池自动出药系统故障";
NETWORK
TITLE =
//补水阀开故障（30秒阀门没开到位）
      A     "补水阀开关";
      L     S5T#30S;
      SD    "补水阀开故障延时";
      A     "补水阀开到位";
      R     "补水阀开故障延时";
      NOP   0;
      NOP   0;
      A     "补水阀开故障延时";
      =     "补水阀故障";
NETWORK
TITLE =
//1号曝气泵运行故障（30秒曝气泵没运行）
      A     "1号曝气泵远程本地";
      A     "曝气泵1号启停";
      L     S5T#30S;
      SD    "1号曝气泵运行故障延时";
      A     "1号曝气泵运行状态";
      R     "1号曝气泵运行故障延时";
      NOP   0;
      NOP   0;
      A     "1号曝气泵运行故障延时";
      =     "1号曝气泵运行故障";
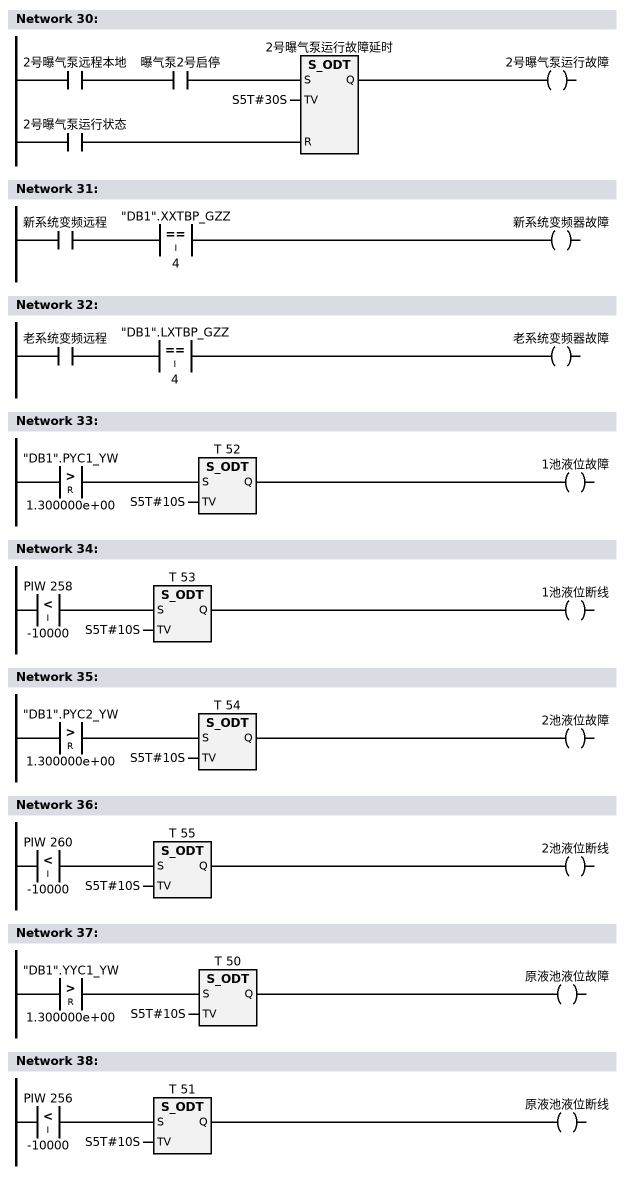
NETWORK
TITLE =
//2号曝气泵运行故障（30秒曝气泵没运行）
      A     "2号曝气泵远程本地";
      A     "曝气泵2号启停";
      L     S5T#30S;
      SD    "2号曝气泵运行故障延时";
      A     "2号曝气泵运行状态";
      R     "2号曝气泵运行故障延时";
      NOP   0;
      NOP   0;
      A     "2号曝气泵运行故障延时";
      =     "2号曝气泵运行故障";
NETWORK
TITLE =
//新系统变频器故障（变频器状态字等于4）
      A     "新系统变频远程";
      A(;
      L     "DB1".XXTBP_GZZ;
      L     4;
      ==I;
      );
      =     "新系统变频器故障";
NETWORK
TITLE =
//老系统变频器故障（变频器状态字等于4）
      A     "老系统变频远程";
      A(;
      L     "DB1".LXTBP_GZZ;
      L     4;
      ==I;
      );
      =     "老系统变频器故障";
NETWORK
TITLE =
//1池液位故障（大于1.3,10秒后）
      A(;
      L     "DB1".PYC1_YW;
      L     1.300000e+00;
      >R;
      );
      L     S5T#10S;
      SD    T 52;
      NOP   0;
      NOP   0;
      NOP   0;
      A     T 52;
      =     "1池液位故障";
NETWORK
TITLE =
//1池液位断线（小于-10000，10秒后）
      A(;
      L     PIW 258;
      L     -10000;
      <I;
      );
      L     S5T#10S;
      SD    T 53;
      NOP   0;
      NOP   0;
      NOP   0;
      A     T 53;
      =     "1池液位断线";
NETWORK
TITLE =
//2池液位故障（大于1.3,10秒后）
      A(;
      L     "DB1".PYC2_YW;
      L     1.300000e+00;
      >R;
      );
      L     S5T#10S;
      SD    T 54;
      NOP   0;
      NOP   0;
      NOP   0;
      A     T 54;
      =     "2池液位故障";
NETWORK
TITLE =
//2池液位断线（小于-10000，10秒后）
      A(;
      L     PIW 260;
      L     -10000;
      <I;
      );
      L     S5T#10S;
      SD    T 55;
      NOP   0;
      NOP   0;
      NOP   0;
      A     T 55;
      =     "2池液位断线";
NETWORK
TITLE =
//原液池液位故障（大于1.3,10秒后）
      A(;
      L     "DB1".YYC1_YW;
      L     1.300000e+00;
      >R;
      );
      L     S5T#10S;
      SD    T 50;
      NOP   0;
      NOP   0;
      NOP   0;
      A     T 50;
      =     "原液池液位故障";
NETWORK
TITLE =
//原液池液位断线（小于-10000，10秒后）
      A(;
      L     PIW 256;
      L     -10000;
      <I;
      );
      L     S5T#10S;
      SD    T 51;
      NOP   0;
      NOP   0;
      NOP   0;
      A     T 51;
      =     "原液池液位断线";
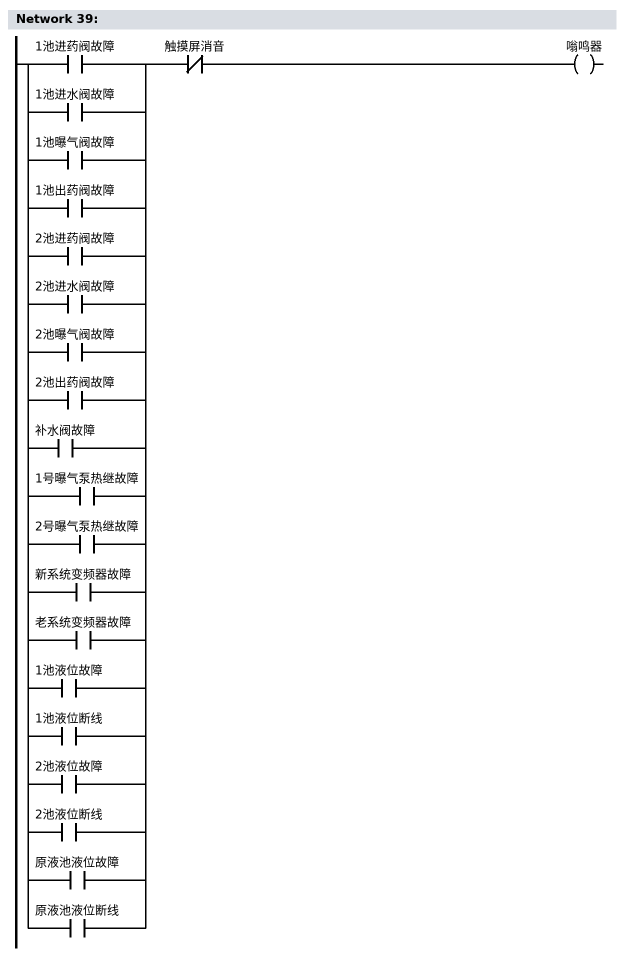
NETWORK
TITLE =
//触摸屏采集的故障点
      A(;
      O     "1池进药阀故障";
      O     "1池进水阀故障";
      O     "1池曝气阀故障";
      O     "1池出药阀故障";
      O     "2池进药阀故障";
      O     "2池进水阀故障";
      O     "2池曝气阀故障";
      O     "2池出药阀故障";
      O     "补水阀故障";
      O     "1号曝气泵热继故障";
      O     "2号曝气泵热继故障";
      O     "新系统变频器故障";
      O     "老系统变频器故障";
      O     "1池液位故障";
      O     "1池液位断线";
      O     "2池液位故障";
      O     "2池液位断线";
      O     "原液池液位故障";
      O     "原液池液位断线";
      );
      AN    "触摸屏消音";
      =     "嗡鸣器";
END_FUNCTION

// FC 40: know-how protected block, not included

// FC 105: know-how protected block, not included

DATA_BLOCK "DB1"	// DB 1
VERSION : 0.1
  STRUCT
   YYC1_YW : REAL ;	//原液池一池液位
   YYC2_YW : REAL ;	//原液池二池液位
   PYC1_YW : REAL ;	//一池液位
   PYC2_YW : REAL ;	//二池液位
   XXTCYLL : REAL ;	//新系统瞬时流量
   lXTCYLL : REAL ;	//老系统瞬时流量
   beiyong1 : REAL ;	//备用
   beiyong2 : REAL ;	//备用
   PYCJYHYW1 : REAL ;	//一池加药后液位设定
   PYCJSHYW1 : REAL ;	//一池加水后液位设定
   PYCJYSDZ : REAL ;	//加药量设定值
   PYCJSSDZ : REAL ;	//加水量设定值
   PYCCSYW : REAL ;	//配药池初始液位
   BQTZSJ : INT ;	//曝气停止时间设定值
   BQYXSJ : INT ;	//曝气运行时间设定值
   BQZQSJ : INT ;	//曝气周期时间设定值
   BQZQJS : INT ;	//一池曝气计时
   BQDSFX : INT ;	//二池曝气计时
   KCYWSD : REAL ;	//空池液位设定
   PYCJYHYW2 : REAL ;	//二池加药后液位设定
   PYCJSHYW2 : REAL ;	//二池加水后液位设定
   YYC1_YWSXSD : REAL ;	//原液池池一液位上限设定
   YYC1_YWXXSD : REAL ;	//原液池池一液位下限设定
   PYC1_YWSXSD : REAL ;	//一池液位上限设定
   PYC1_YWXXSD : REAL ;	//一池液位下限设定
   PYC2_YWSXSD : REAL ;	//二池液位上限设定
   PYC2_YWXXSD : REAL ;	//二池液位下限设定
   XXT_SSLLXXSD : REAL ;	//新系统瞬时流量下限设定
   LXT_SSLLXXSD1 : REAL ;	//老系统瞬时流量下限设定
   XXTBP_GZZ : INT ;	//新系统变频状态
   LXTBP_GZZ : INT ;	//老系统变频状态
   XXTBP_PL : INT ;	//新系统变频频率
   LXTBP_PL : INT ;	//老系统变频频率
  END_STRUCT ;	
BEGIN
   YYC1_YW := 1.210939e+00;
   PYC1_YW := 4.857946e-01;
   PYC2_YW := 1.015706e+00;
   XXTCYLL := 2.864366e+02;
   lXTCYLL := 1.449002e+02;
   PYCJYHYW1 := 2.104565e-01;
   PYCJSHYW1 := 1.010456e+00;
   PYCJYSDZ := 2.500000e-02;
   PYCJSSDZ := 8.000000e-01;
   BQYXSJ := 1;
   BQZQSJ := 180;
   PYCJYHYW2 := 2.119123e-01;
   PYCJSHYW2 := 1.011912e+00;
   XXTBP_GZZ := 1;
   LXTBP_GZZ := 1;
   XXTBP_PL := 33;
   LXTBP_PL := 29;
END_DATA_BLOCK

DATA_BLOCK "DB2"	// DB 2
VERSION : 0.1
  STRUCT
   time0_1 : INT ;
   time0_2 : DINT ;
   time0_3 : DINT ;
   time0_4 : TIME ;
   time0_5 : S5TIME ;
  END_STRUCT ;	
BEGIN
   time0_2 := L#1;
   time0_3 := L#60000;
   time0_4 := T#1M;
   time0_5 := S5T#1M;
END_DATA_BLOCK

ORGANIZATION_BLOCK OB 1
VERSION : 0.1
VAR_TEMP
  TEMP0 : BYTE ;
  TEMP1 : BYTE ;
  TEMP2 : BYTE ;
  TEMP3 : BYTE ;
  TEMP4 : BYTE ;
  TEMP5 : BYTE ;
  TEMP6 : INT ;
  TEMP7 : INT ;
  TEMP8 : INT ;
  TEMP9 : DATE_AND_TIME ;
END_VAR
BEGIN
NETWORK
TITLE =
//打开数据块
      OPN   "DB1";
NETWORK
TITLE =
//打开数据块
      OPN   "DB2";
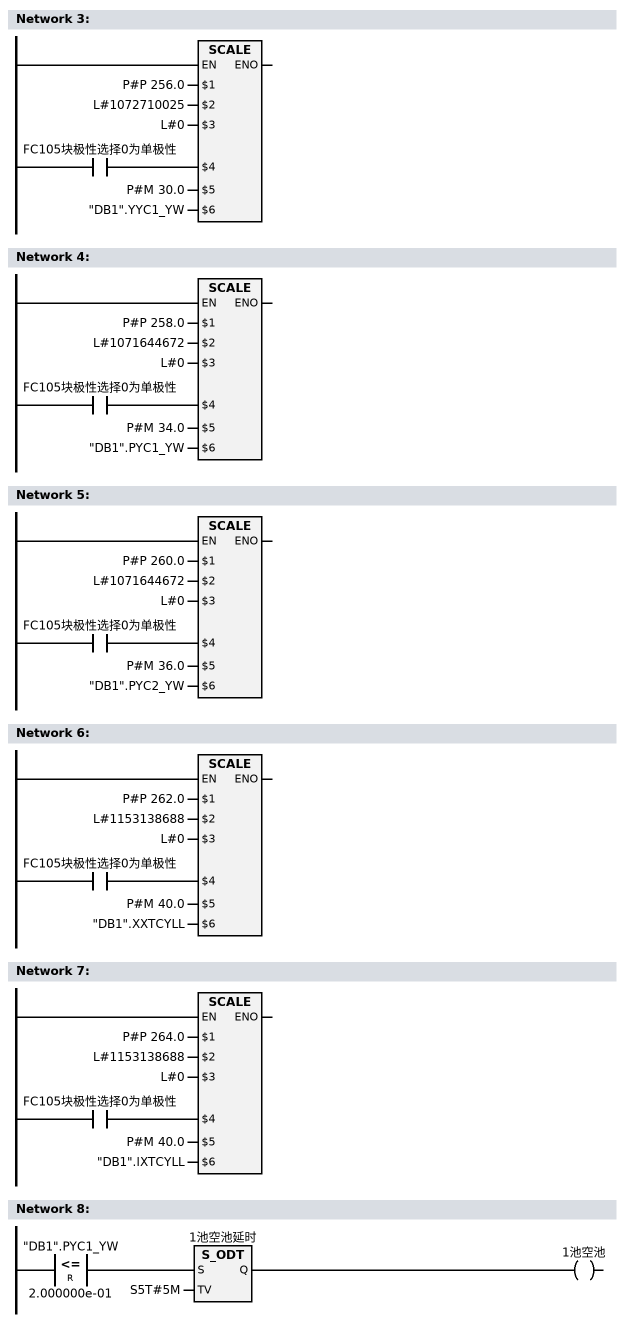
NETWORK
TITLE =
//原液池液位
      A     "FC105块极性选择0为单极性";
      =     L 20.0;
      BLD   103;
      CALL  "SCALE" (
           $1                       := P#P 256.0,
           $2                       := L#1072710025,
           $3                       := L#0,
           $4                       := L 20.0,
           $5                       := P#M 30.0,
           $6                       := "DB1".YYC1_YW);
      NOP   0;
NETWORK
TITLE =
//1#配药池液位
      A     "FC105块极性选择0为单极性";
      =     L 20.0;
      BLD   103;
      CALL  "SCALE" (
           $1                       := P#P 258.0,
           $2                       := L#1071644672,
           $3                       := L#0,
           $4                       := L 20.0,
           $5                       := P#M 34.0,
           $6                       := "DB1".PYC1_YW);
      NOP   0;
NETWORK
TITLE =
//2#配药池液位
      A     "FC105块极性选择0为单极性";
      =     L 20.0;
      BLD   103;
      CALL  "SCALE" (
           $1                       := P#P 260.0,
           $2                       := L#1071644672,
           $3                       := L#0,
           $4                       := L 20.0,
           $5                       := P#M 36.0,
           $6                       := "DB1".PYC2_YW);
      NOP   0;
NETWORK
TITLE =
//新系统瞬时流量
      A     "FC105块极性选择0为单极性";
      =     L 20.0;
      BLD   103;
      CALL  "SCALE" (
           $1                       := P#P 262.0,
           $2                       := L#1153138688,
           $3                       := L#0,
           $4                       := L 20.0,
           $5                       := P#M 40.0,
           $6                       := "DB1".XXTCYLL);
      NOP   0;
NETWORK
TITLE =
//老系统瞬时流量
      A     "FC105块极性选择0为单极性";
      =     L 20.0;
      BLD   103;
      CALL  "SCALE" (
           $1                       := P#P 264.0,
           $2                       := L#1153138688,
           $3                       := L#0,
           $4                       := L 20.0,
           $5                       := P#M 40.0,
           $6                       := "DB1".lXTCYLL);
      NOP   0;
NETWORK
TITLE =
//1#配药池液位小于等于0.2时延时5分钟后，1#配药池空池报警
      A(;
      L     "DB1".PYC1_YW;
      L     2.000000e-01;
      <=R;
      );
      L     S5T#5M;
      SD    "1池空池延时";
      NOP   0;
      NOP   0;
      NOP   0;
      A     "1池空池延时";
      =     "1池空池";
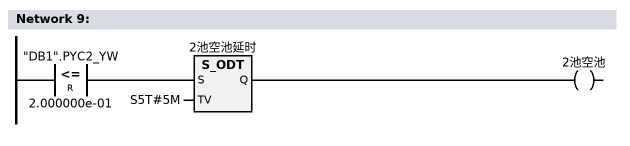
NETWORK
TITLE =
//2#配药池液位小于等于0.2时延时5分钟后，2#配药池空池报警
      A(;
      L     "DB1".PYC2_YW;
      L     2.000000e-01;
      <=R;
      );
      L     S5T#5M;
      SD    "2池空池延时";
      NOP   0;
      NOP   0;
      NOP   0;
      A     "2池空池延时";
      =     "2池空池";
NETWORK
TITLE =
//调用FC块
      UC    "时间转换程序";
NETWORK
TITLE =
//调用FC块
      UC    "报警";
NETWORK
TITLE =
//调用FC块
      UC    "配药";
NETWORK
TITLE =
//调用FC块
      UC    "自动曝气";
NETWORK
TITLE =
//调用FC块
      UC    "自动出药";
NETWORK
TITLE =
//调用FC块
      UC    "计量泵程序";
NETWORK
TITLE =
END_ORGANIZATION_BLOCK

ORGANIZATION_BLOCK "COMPLETE RESTART"	// OB 100
VERSION : 0.1
BEGIN
// (block stored without names or comments; labels and parameter names are numbered)
NETWORK
TITLE =
NETWORK
TITLE =
NETWORK
TITLE =
NETWORK
TITLE =
NETWORK
TITLE =
NETWORK
TITLE =
NETWORK
TITLE =
NETWORK
TITLE =
NETWORK
TITLE =
NETWORK
TITLE =
NETWORK
TITLE =
NETWORK
TITLE =
NETWORK
TITLE =
NETWORK
TITLE =
NETWORK
TITLE =
NETWORK
TITLE =
NETWORK
TITLE =
NETWORK
TITLE =
END_ORGANIZATION_BLOCK

ORGANIZATION_BLOCK "PROG_ERR"	// OB 121
VERSION : 0.1
BEGIN
// (block stored without names or comments; labels and parameter names are numbered)
END_ORGANIZATION_BLOCK
